(* Logix 5000 project; controller reports 1756-L63 rev 20.15; software revision 20.04; part 14 of 52 *)

        [571].time.Day := 11, [571].time.Hour := 15, [571].time.Minute := 59, [571].time.Second := 59, [572].log_data[0].min := 1.0, [572].log_data[0].max := 1.0, [572].log_data[0].total := 300.0, [572].log_data[0].time := 300.0, [572].log_data[0].valid := 1, [572].log_data[1].valid := 1, [572].log_data[2].valid := 1, [572].log_data[3].valid := 1, [572].log_data[4].valid := 1, [572].log_data[5].valid := 1, [572].log_data[6].valid := 1, [572].log_data[7].valid := 1, [572].log_data[8].valid := 1, [572].log_data[9].valid := 1, [572].log_data[10].valid := 1, [572].log_data[11].valid := 1, [572].log_data[12].valid := 1, [572].log_data[13].valid := 1, [572].log_data[14].valid := 1, [572].log_data[15].valid := 1, [572].log_data[16].valid := 1, [572].log_data[17].valid := 1, [572].log_data[18].valid := 1, [572].log_data[19].valid := 1, [572].time.Year := 2023, [572].time.Month := 1, [572].time.Day := 11, [572].time.Hour := 16, [572].time.Minute := 4, [572].time.Second := 59, [573].log_data[0].min := 1.0, [573].log_data[0].max := 1.0, [573].log_data[0].total := 300.0, [573].log_data[0].time := 300.0, [573].log_data[0].minminute := 5, [573].log_data[0].maxminute := 5, [573].log_data[0].valid := 1, [573].log_data[1].valid := 1, [573].log_data[2].valid := 1, [573].log_data[3].valid := 1, [573].log_data[4].valid := 1, [573].log_data[5].valid := 1, [573].log_data[6].valid := 1, [573].log_data[7].valid := 1, [573].log_data[8].valid := 1, [573].log_data[9].valid := 1, [573].log_data[10].valid := 1, [573].log_data[11].valid := 1, [573].log_data[12].valid := 1, [573].log_data[13].valid := 1, [573].log_data[14].valid := 1, [573].log_data[15].valid := 1, [573].log_data[16].valid := 1, [573].log_data[17].valid := 1, [573].log_data[18].valid := 1, [573].log_data[19].valid := 1,
        [573].time.Year := 2023, [573].time.Month := 1, [573].time.Day := 11, [573].time.Hour := 16, [573].time.Minute := 9, [573].time.Second := 59, [574].log_data[0].min := 1.0, [574].log_data[0].max := 1.0, [574].log_data[0].total := 300.0, [574].log_data[0].time := 300.0, [574].log_data[0].minminute := 10, [574].log_data[0].maxminute := 10, [574].log_data[0].valid := 1, [574].log_data[1].valid := 1, [574].log_data[2].valid := 1, [574].log_data[3].valid := 1, [574].log_data[4].valid := 1, [574].log_data[5].valid := 1, [574].log_data[6].valid := 1, [574].log_data[7].valid := 1, [574].log_data[8].valid := 1, [574].log_data[9].valid := 1, [574].log_data[10].valid := 1, [574].log_data[11].valid := 1, [574].log_data[12].valid := 1, [574].log_data[13].valid := 1, [574].log_data[14].valid := 1, [574].log_data[15].valid := 1, [574].log_data[16].valid := 1, [574].log_data[17].valid := 1, [574].log_data[18].valid := 1, [574].log_data[19].valid := 1, [574].time.Year := 2023, [574].time.Month := 1, [574].time.Day := 11, [574].time.Hour := 16, [574].time.Minute := 14, [574].time.Second := 59, [575].log_data[0].min := 1.0, [575].log_data[0].max := 1.0, [575].log_data[0].total := 300.0, [575].log_data[0].time := 300.0, [575].log_data[0].minminute := 15, [575].log_data[0].maxminute := 15, [575].log_data[0].valid := 1, [575].log_data[1].valid := 1, [575].log_data[2].valid := 1, [575].log_data[3].valid := 1, [575].log_data[4].valid := 1, [575].log_data[5].valid := 1, [575].log_data[6].valid := 1, [575].log_data[7].valid := 1, [575].log_data[8].valid := 1, [575].log_data[9].valid := 1, [575].log_data[10].valid := 1, [575].log_data[11].valid := 1, [575].log_data[12].valid := 1, [575].log_data[13].valid := 1, [575].log_data[14].valid := 1, [575].log_data[15].valid := 1,
        [575].log_data[16].valid := 1, [575].log_data[17].valid := 1, [575].log_data[18].valid := 1, [575].log_data[19].valid := 1, [575].time.Year := 2023, [575].time.Month := 1, [575].time.Day := 11, [575].time.Hour := 16, [575].time.Minute := 19, [575].time.Second := 59, [576].log_data[0].min := 1.0, [576].log_data[0].max := 1.0, [576].log_data[0].total := 300.0, [576].log_data[0].time := 300.0, [576].log_data[0].minminute := 20, [576].log_data[0].maxminute := 20, [576].log_data[0].valid := 1, [576].log_data[1].valid := 1, [576].log_data[2].valid := 1, [576].log_data[3].valid := 1, [576].log_data[4].valid := 1, [576].log_data[5].valid := 1, [576].log_data[6].valid := 1, [576].log_data[7].valid := 1, [576].log_data[8].valid := 1, [576].log_data[9].valid := 1, [576].log_data[10].valid := 1, [576].log_data[11].valid := 1, [576].log_data[12].valid := 1, [576].log_data[13].valid := 1, [576].log_data[14].valid := 1, [576].log_data[15].valid := 1, [576].log_data[16].valid := 1, [576].log_data[17].valid := 1, [576].log_data[18].valid := 1, [576].log_data[19].valid := 1, [576].time.Year := 2023, [576].time.Month := 1, [576].time.Day := 11, [576].time.Hour := 16, [576].time.Minute := 24, [576].time.Second := 59, [577].log_data[0].min := 1.0, [577].log_data[0].max := 1.0, [577].log_data[0].total := 300.0, [577].log_data[0].time := 300.0, [577].log_data[0].minminute := 25, [577].log_data[0].maxminute := 25, [577].log_data[0].valid := 1, [577].log_data[1].valid := 1, [577].log_data[2].valid := 1, [577].log_data[3].valid := 1, [577].log_data[4].valid := 1, [577].log_data[5].valid := 1, [577].log_data[6].valid := 1, [577].log_data[7].valid := 1, [577].log_data[8].valid := 1, [577].log_data[9].valid := 1, [577].log_data[10].valid := 1, [577].log_data[11].valid := 1,
        [577].log_data[12].valid := 1, [577].log_data[13].valid := 1, [577].log_data[14].valid := 1, [577].log_data[15].valid := 1, [577].log_data[16].valid := 1, [577].log_data[17].valid := 1, [577].log_data[18].valid := 1, [577].log_data[19].valid := 1, [577].time.Year := 2023, [577].time.Month := 1, [577].time.Day := 11, [577].time.Hour := 16, [577].time.Minute := 29, [577].time.Second := 59, [578].log_data[0].min := 1.0, [578].log_data[0].max := 1.0, [578].log_data[0].total := 300.0, [578].log_data[0].time := 300.0, [578].log_data[0].minminute := 30, [578].log_data[0].maxminute := 30, [578].log_data[0].valid := 1, [578].log_data[1].valid := 1, [578].log_data[2].valid := 1, [578].log_data[3].valid := 1, [578].log_data[4].valid := 1, [578].log_data[5].valid := 1, [578].log_data[6].valid := 1, [578].log_data[7].valid := 1, [578].log_data[8].valid := 1, [578].log_data[9].valid := 1, [578].log_data[10].valid := 1, [578].log_data[11].valid := 1, [578].log_data[12].valid := 1, [578].log_data[13].valid := 1, [578].log_data[14].valid := 1, [578].log_data[15].valid := 1, [578].log_data[16].valid := 1, [578].log_data[17].valid := 1, [578].log_data[18].valid := 1, [578].log_data[19].valid := 1, [578].time.Year := 2023, [578].time.Month := 1, [578].time.Day := 11, [578].time.Hour := 16, [578].time.Minute := 34, [578].time.Second := 59, [579].log_data[0].min := 1.0, [579].log_data[0].max := 1.0, [579].log_data[0].total := 300.0, [579].log_data[0].time := 300.0, [579].log_data[0].minminute := 35, [579].log_data[0].maxminute := 35, [579].log_data[0].valid := 1, [579].log_data[1].valid := 1, [579].log_data[2].valid := 1, [579].log_data[3].valid := 1, [579].log_data[4].valid := 1, [579].log_data[5].valid := 1, [579].log_data[6].valid := 1, [579].log_data[7].valid := 1,
        [579].log_data[8].valid := 1, [579].log_data[9].valid := 1, [579].log_data[10].valid := 1, [579].log_data[11].valid := 1, [579].log_data[12].valid := 1, [579].log_data[13].valid := 1, [579].log_data[14].valid := 1, [579].log_data[15].valid := 1, [579].log_data[16].valid := 1, [579].log_data[17].valid := 1, [579].log_data[18].valid := 1, [579].log_data[19].valid := 1, [579].time.Year := 2023, [579].time.Month := 1, [579].time.Day := 11, [579].time.Hour := 16, [579].time.Minute := 39, [579].time.Second := 59, [580].log_data[0].min := 1.0, [580].log_data[0].max := 1.0, [580].log_data[0].total := 300.0, [580].log_data[0].time := 300.0, [580].log_data[0].minminute := 40, [580].log_data[0].maxminute := 40, [580].log_data[0].valid := 1, [580].log_data[1].valid := 1, [580].log_data[2].valid := 1, [580].log_data[3].valid := 1, [580].log_data[4].valid := 1, [580].log_data[5].valid := 1, [580].log_data[6].valid := 1, [580].log_data[7].valid := 1, [580].log_data[8].valid := 1, [580].log_data[9].valid := 1, [580].log_data[10].valid := 1, [580].log_data[11].valid := 1, [580].log_data[12].valid := 1, [580].log_data[13].valid := 1, [580].log_data[14].valid := 1, [580].log_data[15].valid := 1, [580].log_data[16].valid := 1, [580].log_data[17].valid := 1, [580].log_data[18].valid := 1, [580].log_data[19].valid := 1, [580].time.Year := 2023, [580].time.Month := 1, [580].time.Day := 11, [580].time.Hour := 16, [580].time.Minute := 44, [580].time.Second := 59, [581].log_data[0].min := 1.0, [581].log_data[0].max := 1.0, [581].log_data[0].total := 300.0, [581].log_data[0].time := 300.0, [581].log_data[0].minminute := 45, [581].log_data[0].maxminute := 45, [581].log_data[0].valid := 1, [581].log_data[1].valid := 1, [581].log_data[2].valid := 1, [581].log_data[3].valid := 1,
        [581].log_data[4].valid := 1, [581].log_data[5].valid := 1, [581].log_data[6].valid := 1, [581].log_data[7].valid := 1, [581].log_data[8].valid := 1, [581].log_data[9].valid := 1, [581].log_data[10].valid := 1, [581].log_data[11].valid := 1, [581].log_data[12].valid := 1, [581].log_data[13].valid := 1, [581].log_data[14].valid := 1, [581].log_data[15].valid := 1, [581].log_data[16].valid := 1, [581].log_data[17].valid := 1, [581].log_data[18].valid := 1, [581].log_data[19].valid := 1, [581].time.Year := 2023, [581].time.Month := 1, [581].time.Day := 11, [581].time.Hour := 16, [581].time.Minute := 49, [581].time.Second := 59, [582].log_data[0].min := 1.0, [582].log_data[0].max := 1.0, [582].log_data[0].total := 300.0, [582].log_data[0].time := 300.0, [582].log_data[0].minminute := 50, [582].log_data[0].maxminute := 50, [582].log_data[0].valid := 1, [582].log_data[1].valid := 1, [582].log_data[2].valid := 1, [582].log_data[3].valid := 1, [582].log_data[4].valid := 1, [582].log_data[5].valid := 1, [582].log_data[6].valid := 1, [582].log_data[7].valid := 1, [582].log_data[8].valid := 1, [582].log_data[9].valid := 1, [582].log_data[10].valid := 1, [582].log_data[11].valid := 1, [582].log_data[12].valid := 1, [582].log_data[13].valid := 1, [582].log_data[14].valid := 1, [582].log_data[15].valid := 1, [582].log_data[16].valid := 1, [582].log_data[17].valid := 1, [582].log_data[18].valid := 1, [582].log_data[19].valid := 1, [582].time.Year := 2023, [582].time.Month := 1, [582].time.Day := 11, [582].time.Hour := 16, [582].time.Minute := 54, [582].time.Second := 59, [583].log_data[0].min := 1.0, [583].log_data[0].max := 1.0, [583].log_data[0].total := 300.0, [583].log_data[0].time := 300.0, [583].log_data[0].minminute := 55, [583].log_data[0].maxminute := 55,
        [583].log_data[0].valid := 1, [583].log_data[1].valid := 1, [583].log_data[2].valid := 1, [583].log_data[3].valid := 1, [583].log_data[4].valid := 1, [583].log_data[5].valid := 1, [583].log_data[6].valid := 1, [583].log_data[7].valid := 1, [583].log_data[8].valid := 1, [583].log_data[9].valid := 1, [583].log_data[10].valid := 1, [583].log_data[11].valid := 1, [583].log_data[12].valid := 1, [583].log_data[13].valid := 1, [583].log_data[14].valid := 1, [583].log_data[15].valid := 1, [583].log_data[16].valid := 1, [583].log_data[17].valid := 1, [583].log_data[18].valid := 1, [583].log_data[19].valid := 1, [583].time.Year := 2023, [583].time.Month := 1, [583].time.Day := 11, [583].time.Hour := 16, [583].time.Minute := 59, [583].time.Second := 59, [584].log_data[0].min := 1.0, [584].log_data[0].max := 1.0, [584].log_data[0].total := 300.0, [584].log_data[0].time := 300.0, [584].log_data[0].valid := 1, [584].log_data[1].valid := 1, [584].log_data[2].valid := 1, [584].log_data[3].valid := 1, [584].log_data[4].valid := 1, [584].log_data[5].valid := 1, [584].log_data[6].valid := 1, [584].log_data[7].valid := 1, [584].log_data[8].valid := 1, [584].log_data[9].valid := 1, [584].log_data[10].valid := 1, [584].log_data[11].valid := 1, [584].log_data[12].valid := 1, [584].log_data[13].valid := 1, [584].log_data[14].valid := 1, [584].log_data[15].valid := 1, [584].log_data[16].valid := 1, [584].log_data[17].valid := 1, [584].log_data[18].valid := 1, [584].log_data[19].valid := 1, [584].time.Year := 2023, [584].time.Month := 1, [584].time.Day := 11, [584].time.Hour := 17, [584].time.Minute := 4, [584].time.Second := 59, [585].log_data[0].min := 1.0, [585].log_data[0].max := 1.0, [585].log_data[0].total := 300.0, [585].log_data[0].time := 300.0,
        [585].log_data[0].minminute := 5, [585].log_data[0].maxminute := 5, [585].log_data[0].valid := 1, [585].log_data[1].valid := 1, [585].log_data[2].valid := 1, [585].log_data[3].valid := 1, [585].log_data[4].valid := 1, [585].log_data[5].valid := 1, [585].log_data[6].valid := 1, [585].log_data[7].valid := 1, [585].log_data[8].valid := 1, [585].log_data[9].valid := 1, [585].log_data[10].valid := 1, [585].log_data[11].valid := 1, [585].log_data[12].valid := 1, [585].log_data[13].valid := 1, [585].log_data[14].valid := 1, [585].log_data[15].valid := 1, [585].log_data[16].valid := 1, [585].log_data[17].valid := 1, [585].log_data[18].valid := 1, [585].log_data[19].valid := 1, [585].time.Year := 2023, [585].time.Month := 1, [585].time.Day := 11, [585].time.Hour := 17, [585].time.Minute := 9, [585].time.Second := 59, [586].log_data[0].min := 1.0, [586].log_data[0].max := 1.0, [586].log_data[0].total := 300.0, [586].log_data[0].time := 300.0, [586].log_data[0].minminute := 10, [586].log_data[0].maxminute := 10, [586].log_data[0].valid := 1, [586].log_data[1].valid := 1, [586].log_data[2].valid := 1, [586].log_data[3].valid := 1, [586].log_data[4].valid := 1, [586].log_data[5].valid := 1, [586].log_data[6].valid := 1, [586].log_data[7].valid := 1, [586].log_data[8].valid := 1, [586].log_data[9].valid := 1, [586].log_data[10].valid := 1, [586].log_data[11].valid := 1, [586].log_data[12].valid := 1, [586].log_data[13].valid := 1, [586].log_data[14].valid := 1, [586].log_data[15].valid := 1, [586].log_data[16].valid := 1, [586].log_data[17].valid := 1, [586].log_data[18].valid := 1, [586].log_data[19].valid := 1, [586].time.Year := 2023, [586].time.Month := 1, [586].time.Day := 11, [586].time.Hour := 17, [586].time.Minute := 14, [586].time.Second := 59,
        [587].log_data[0].min := 1.0, [587].log_data[0].max := 1.0, [587].log_data[0].total := 300.0, [587].log_data[0].time := 300.0, [587].log_data[0].minminute := 15, [587].log_data[0].maxminute := 15, [587].log_data[0].valid := 1, [587].log_data[1].valid := 1, [587].log_data[2].valid := 1, [587].log_data[3].valid := 1, [587].log_data[4].valid := 1, [587].log_data[5].valid := 1, [587].log_data[6].valid := 1, [587].log_data[7].valid := 1, [587].log_data[8].valid := 1, [587].log_data[9].valid := 1, [587].log_data[10].valid := 1, [587].log_data[11].valid := 1, [587].log_data[12].valid := 1, [587].log_data[13].valid := 1, [587].log_data[14].valid := 1, [587].log_data[15].valid := 1, [587].log_data[16].valid := 1, [587].log_data[17].valid := 1, [587].log_data[18].valid := 1, [587].log_data[19].valid := 1, [587].time.Year := 2023, [587].time.Month := 1, [587].time.Day := 11, [587].time.Hour := 17, [587].time.Minute := 19, [587].time.Second := 59, [588].log_data[0].min := 1.0, [588].log_data[0].max := 1.0, [588].log_data[0].total := 300.0, [588].log_data[0].time := 300.0, [588].log_data[0].minminute := 20, [588].log_data[0].maxminute := 20, [588].log_data[0].valid := 1, [588].log_data[1].valid := 1, [588].log_data[2].valid := 1, [588].log_data[3].valid := 1, [588].log_data[4].valid := 1, [588].log_data[5].valid := 1, [588].log_data[6].valid := 1, [588].log_data[7].valid := 1, [588].log_data[8].valid := 1, [588].log_data[9].valid := 1, [588].log_data[10].valid := 1, [588].log_data[11].valid := 1, [588].log_data[12].valid := 1, [588].log_data[13].valid := 1, [588].log_data[14].valid := 1, [588].log_data[15].valid := 1, [588].log_data[16].valid := 1, [588].log_data[17].valid := 1, [588].log_data[18].valid := 1, [588].log_data[19].valid := 1, [588].time.Year := 2023, [588].time.Month := 1,
        [588].time.Day := 11, [588].time.Hour := 17, [588].time.Minute := 24, [588].time.Second := 59, [589].log_data[0].min := 1.0, [589].log_data[0].max := 1.0, [589].log_data[0].total := 300.0, [589].log_data[0].time := 300.0, [589].log_data[0].minminute := 25, [589].log_data[0].maxminute := 25, [589].log_data[0].valid := 1, [589].log_data[1].valid := 1, [589].log_data[2].valid := 1, [589].log_data[3].valid := 1, [589].log_data[4].valid := 1, [589].log_data[5].valid := 1, [589].log_data[6].valid := 1, [589].log_data[7].valid := 1, [589].log_data[8].valid := 1, [589].log_data[9].valid := 1, [589].log_data[10].valid := 1, [589].log_data[11].valid := 1, [589].log_data[12].valid := 1, [589].log_data[13].valid := 1, [589].log_data[14].valid := 1, [589].log_data[15].valid := 1, [589].log_data[16].valid := 1, [589].log_data[17].valid := 1, [589].log_data[18].valid := 1, [589].log_data[19].valid := 1, [589].time.Year := 2023, [589].time.Month := 1, [589].time.Day := 11, [589].time.Hour := 17, [589].time.Minute := 29, [589].time.Second := 59, [590].log_data[0].min := 1.0, [590].log_data[0].max := 1.0, [590].log_data[0].total := 300.0, [590].log_data[0].time := 300.0, [590].log_data[0].minminute := 30, [590].log_data[0].maxminute := 30, [590].log_data[0].valid := 1, [590].log_data[1].valid := 1, [590].log_data[2].valid := 1, [590].log_data[3].valid := 1, [590].log_data[4].valid := 1, [590].log_data[5].valid := 1, [590].log_data[6].valid := 1, [590].log_data[7].valid := 1, [590].log_data[8].valid := 1, [590].log_data[9].valid := 1, [590].log_data[10].valid := 1, [590].log_data[11].valid := 1, [590].log_data[12].valid := 1, [590].log_data[13].valid := 1, [590].log_data[14].valid := 1, [590].log_data[15].valid := 1, [590].log_data[16].valid := 1, [590].log_data[17].valid := 1,
        [590].log_data[18].valid := 1, [590].log_data[19].valid := 1, [590].time.Year := 2023, [590].time.Month := 1, [590].time.Day := 11, [590].time.Hour := 17, [590].time.Minute := 34, [590].time.Second := 59, [591].log_data[0].min := 1.0, [591].log_data[0].max := 1.0, [591].log_data[0].total := 300.0, [591].log_data[0].time := 300.0, [591].log_data[0].minminute := 35, [591].log_data[0].maxminute := 35, [591].log_data[0].valid := 1, [591].log_data[1].valid := 1, [591].log_data[2].valid := 1, [591].log_data[3].valid := 1, [591].log_data[4].valid := 1, [591].log_data[5].valid := 1, [591].log_data[6].valid := 1, [591].log_data[7].valid := 1, [591].log_data[8].valid := 1, [591].log_data[9].valid := 1, [591].log_data[10].valid := 1, [591].log_data[11].valid := 1, [591].log_data[12].valid := 1, [591].log_data[13].valid := 1, [591].log_data[14].valid := 1, [591].log_data[15].valid := 1, [591].log_data[16].valid := 1, [591].log_data[17].valid := 1, [591].log_data[18].valid := 1, [591].log_data[19].valid := 1, [591].time.Year := 2023, [591].time.Month := 1, [591].time.Day := 11, [591].time.Hour := 17, [591].time.Minute := 39, [591].time.Second := 59, [592].log_data[0].min := 1.0, [592].log_data[0].max := 1.0, [592].log_data[0].total := 300.0, [592].log_data[0].time := 300.0, [592].log_data[0].minminute := 40, [592].log_data[0].maxminute := 40, [592].log_data[0].valid := 1, [592].log_data[1].valid := 1, [592].log_data[2].valid := 1, [592].log_data[3].valid := 1, [592].log_data[4].valid := 1, [592].log_data[5].valid := 1, [592].log_data[6].valid := 1, [592].log_data[7].valid := 1, [592].log_data[8].valid := 1, [592].log_data[9].valid := 1, [592].log_data[10].valid := 1, [592].log_data[11].valid := 1, [592].log_data[12].valid := 1, [592].log_data[13].valid := 1,
        [592].log_data[14].valid := 1, [592].log_data[15].valid := 1, [592].log_data[16].valid := 1, [592].log_data[17].valid := 1, [592].log_data[18].valid := 1, [592].log_data[19].valid := 1, [592].time.Year := 2023, [592].time.Month := 1, [592].time.Day := 11, [592].time.Hour := 17, [592].time.Minute := 44, [592].time.Second := 59, [593].log_data[0].min := 1.0, [593].log_data[0].max := 1.0, [593].log_data[0].total := 300.0, [593].log_data[0].time := 300.0, [593].log_data[0].minminute := 45, [593].log_data[0].maxminute := 45, [593].log_data[0].valid := 1, [593].log_data[1].valid := 1, [593].log_data[2].valid := 1, [593].log_data[3].valid := 1, [593].log_data[4].valid := 1, [593].log_data[5].valid := 1, [593].log_data[6].valid := 1, [593].log_data[7].valid := 1, [593].log_data[8].valid := 1, [593].log_data[9].valid := 1, [593].log_data[10].valid := 1, [593].log_data[11].valid := 1, [593].log_data[12].valid := 1, [593].log_data[13].valid := 1, [593].log_data[14].valid := 1, [593].log_data[15].valid := 1, [593].log_data[16].valid := 1, [593].log_data[17].valid := 1, [593].log_data[18].valid := 1, [593].log_data[19].valid := 1, [593].time.Year := 2023, [593].time.Month := 1, [593].time.Day := 11, [593].time.Hour := 17, [593].time.Minute := 49, [593].time.Second := 59, [594].log_data[0].min := 1.0, [594].log_data[0].max := 1.0, [594].log_data[0].total := 300.0, [594].log_data[0].time := 300.0, [594].log_data[0].minminute := 50, [594].log_data[0].maxminute := 50, [594].log_data[0].valid := 1, [594].log_data[1].valid := 1, [594].log_data[2].valid := 1, [594].log_data[3].valid := 1, [594].log_data[4].valid := 1, [594].log_data[5].valid := 1, [594].log_data[6].valid := 1, [594].log_data[7].valid := 1, [594].log_data[8].valid := 1, [594].log_data[9].valid := 1,
        [594].log_data[10].valid := 1, [594].log_data[11].valid := 1, [594].log_data[12].valid := 1, [594].log_data[13].valid := 1, [594].log_data[14].valid := 1, [594].log_data[15].valid := 1, [594].log_data[16].valid := 1, [594].log_data[17].valid := 1, [594].log_data[18].valid := 1, [594].log_data[19].valid := 1, [594].time.Year := 2023, [594].time.Month := 1, [594].time.Day := 11, [594].time.Hour := 17, [594].time.Minute := 54, [594].time.Second := 59, [595].log_data[0].min := 1.0, [595].log_data[0].max := 1.0, [595].log_data[0].total := 300.0, [595].log_data[0].time := 300.0, [595].log_data[0].minminute := 55, [595].log_data[0].maxminute := 55, [595].log_data[0].valid := 1, [595].log_data[1].valid := 1, [595].log_data[2].valid := 1, [595].log_data[3].valid := 1, [595].log_data[4].valid := 1, [595].log_data[5].valid := 1, [595].log_data[6].valid := 1, [595].log_data[7].valid := 1, [595].log_data[8].valid := 1, [595].log_data[9].valid := 1, [595].log_data[10].valid := 1, [595].log_data[11].valid := 1, [595].log_data[12].valid := 1, [595].log_data[13].valid := 1, [595].log_data[14].valid := 1, [595].log_data[15].valid := 1, [595].log_data[16].valid := 1, [595].log_data[17].valid := 1, [595].log_data[18].valid := 1, [595].log_data[19].valid := 1, [595].time.Year := 2023, [595].time.Month := 1, [595].time.Day := 11, [595].time.Hour := 17, [595].time.Minute := 59, [595].time.Second := 59, [596].log_data[0].min := 1.0, [596].log_data[0].max := 1.0, [596].log_data[0].total := 300.0, [596].log_data[0].time := 300.0, [596].log_data[0].valid := 1, [596].log_data[1].valid := 1, [596].log_data[2].valid := 1, [596].log_data[3].valid := 1, [596].log_data[4].valid := 1, [596].log_data[5].valid := 1, [596].log_data[6].valid := 1, [596].log_data[7].valid := 1,
        [596].log_data[8].valid := 1, [596].log_data[9].valid := 1, [596].log_data[10].valid := 1, [596].log_data[11].valid := 1, [596].log_data[12].valid := 1, [596].log_data[13].valid := 1, [596].log_data[14].valid := 1, [596].log_data[15].valid := 1, [596].log_data[16].valid := 1, [596].log_data[17].valid := 1, [596].log_data[18].valid := 1, [596].log_data[19].valid := 1, [596].time.Year := 2023, [596].time.Month := 1, [596].time.Day := 11, [596].time.Hour := 18, [596].time.Minute := 4, [596].time.Second := 59, [597].log_data[0].min := 1.0, [597].log_data[0].max := 1.0, [597].log_data[0].total := 300.0, [597].log_data[0].time := 300.0, [597].log_data[0].minminute := 5, [597].log_data[0].maxminute := 5, [597].log_data[0].valid := 1, [597].log_data[1].valid := 1, [597].log_data[2].valid := 1, [597].log_data[3].valid := 1, [597].log_data[4].valid := 1, [597].log_data[5].valid := 1, [597].log_data[6].valid := 1, [597].log_data[7].valid := 1, [597].log_data[8].valid := 1, [597].log_data[9].valid := 1, [597].log_data[10].valid := 1, [597].log_data[11].valid := 1, [597].log_data[12].valid := 1, [597].log_data[13].valid := 1, [597].log_data[14].valid := 1, [597].log_data[15].valid := 1, [597].log_data[16].valid := 1, [597].log_data[17].valid := 1, [597].log_data[18].valid := 1, [597].log_data[19].valid := 1, [597].time.Year := 2023, [597].time.Month := 1, [597].time.Day := 11, [597].time.Hour := 18, [597].time.Minute := 9, [597].time.Second := 59, [598].log_data[0].min := 1.0, [598].log_data[0].max := 1.0, [598].log_data[0].total := 300.0, [598].log_data[0].time := 300.0, [598].log_data[0].minminute := 10, [598].log_data[0].maxminute := 10, [598].log_data[0].valid := 1, [598].log_data[1].valid := 1, [598].log_data[2].valid := 1, [598].log_data[3].valid := 1,
        [598].log_data[4].valid := 1, [598].log_data[5].valid := 1, [598].log_data[6].valid := 1, [598].log_data[7].valid := 1, [598].log_data[8].valid := 1, [598].log_data[9].valid := 1, [598].log_data[10].valid := 1, [598].log_data[11].valid := 1, [598].log_data[12].valid := 1, [598].log_data[13].valid := 1, [598].log_data[14].valid := 1, [598].log_data[15].valid := 1, [598].log_data[16].valid := 1, [598].log_data[17].valid := 1, [598].log_data[18].valid := 1, [598].log_data[19].valid := 1, [598].time.Year := 2023, [598].time.Month := 1, [598].time.Day := 11, [598].time.Hour := 18, [598].time.Minute := 14, [598].time.Second := 59, [599].log_data[0].min := 1.0, [599].log_data[0].max := 1.0, [599].log_data[0].total := 300.0, [599].log_data[0].time := 300.0, [599].log_data[0].minminute := 15, [599].log_data[0].maxminute := 15, [599].log_data[0].valid := 1, [599].log_data[1].valid := 1, [599].log_data[2].valid := 1, [599].log_data[3].valid := 1, [599].log_data[4].valid := 1, [599].log_data[5].valid := 1, [599].log_data[6].valid := 1, [599].log_data[7].valid := 1, [599].log_data[8].valid := 1, [599].log_data[9].valid := 1, [599].log_data[10].valid := 1, [599].log_data[11].valid := 1, [599].log_data[12].valid := 1, [599].log_data[13].valid := 1, [599].log_data[14].valid := 1, [599].log_data[15].valid := 1, [599].log_data[16].valid := 1, [599].log_data[17].valid := 1, [599].log_data[18].valid := 1, [599].log_data[19].valid := 1, [599].time.Year := 2023, [599].time.Month := 1, [599].time.Day := 11, [599].time.Hour := 18, [599].time.Minute := 19, [599].time.Second := 59, [600].log_data[0].min := 1.0, [600].log_data[0].max := 1.0, [600].log_data[0].total := 300.0, [600].log_data[0].time := 300.0, [600].log_data[0].minminute := 20, [600].log_data[0].maxminute := 20,
        [600].log_data[0].valid := 1, [600].log_data[1].valid := 1, [600].log_data[2].valid := 1, [600].log_data[3].valid := 1, [600].log_data[4].valid := 1, [600].log_data[5].valid := 1, [600].log_data[6].valid := 1, [600].log_data[7].valid := 1, [600].log_data[8].valid := 1, [600].log_data[9].valid := 1, [600].log_data[10].valid := 1, [600].log_data[11].valid := 1, [600].log_data[12].valid := 1, [600].log_data[13].valid := 1, [600].log_data[14].valid := 1, [600].log_data[15].valid := 1, [600].log_data[16].valid := 1, [600].log_data[17].valid := 1, [600].log_data[18].valid := 1, [600].log_data[19].valid := 1, [600].time.Year := 2023, [600].time.Month := 1, [600].time.Day := 11, [600].time.Hour := 18, [600].time.Minute := 24, [600].time.Second := 59, [601].log_data[0].min := 1.0, [601].log_data[0].max := 1.0, [601].log_data[0].total := 300.0, [601].log_data[0].time := 300.0, [601].log_data[0].minminute := 25, [601].log_data[0].maxminute := 25, [601].log_data[0].valid := 1, [601].log_data[1].valid := 1, [601].log_data[2].valid := 1, [601].log_data[3].valid := 1, [601].log_data[4].valid := 1, [601].log_data[5].valid := 1, [601].log_data[6].valid := 1, [601].log_data[7].valid := 1, [601].log_data[8].valid := 1, [601].log_data[9].valid := 1, [601].log_data[10].valid := 1, [601].log_data[11].valid := 1, [601].log_data[12].valid := 1, [601].log_data[13].valid := 1, [601].log_data[14].valid := 1, [601].log_data[15].valid := 1, [601].log_data[16].valid := 1, [601].log_data[17].valid := 1, [601].log_data[18].valid := 1, [601].log_data[19].valid := 1, [601].time.Year := 2023, [601].time.Month := 1, [601].time.Day := 11, [601].time.Hour := 18, [601].time.Minute := 29, [601].time.Second := 59, [602].log_data[0].min := 1.0, [602].log_data[0].max := 1.0,
        [602].log_data[0].total := 300.0, [602].log_data[0].time := 300.0, [602].log_data[0].minminute := 30, [602].log_data[0].maxminute := 30, [602].log_data[0].valid := 1, [602].log_data[1].valid := 1, [602].log_data[2].valid := 1, [602].log_data[3].valid := 1, [602].log_data[4].valid := 1, [602].log_data[5].valid := 1, [602].log_data[6].valid := 1, [602].log_data[7].valid := 1, [602].log_data[8].valid := 1, [602].log_data[9].valid := 1, [602].log_data[10].valid := 1, [602].log_data[11].valid := 1, [602].log_data[12].valid := 1, [602].log_data[13].valid := 1, [602].log_data[14].valid := 1, [602].log_data[15].valid := 1, [602].log_data[16].valid := 1, [602].log_data[17].valid := 1, [602].log_data[18].valid := 1, [602].log_data[19].valid := 1, [602].time.Year := 2023, [602].time.Month := 1, [602].time.Day := 11, [602].time.Hour := 18, [602].time.Minute := 34, [602].time.Second := 59, [603].log_data[0].min := 1.0, [603].log_data[0].max := 1.0, [603].log_data[0].total := 300.0, [603].log_data[0].time := 300.0, [603].log_data[0].minminute := 35, [603].log_data[0].maxminute := 35, [603].log_data[0].valid := 1, [603].log_data[1].valid := 1, [603].log_data[2].valid := 1, [603].log_data[3].valid := 1, [603].log_data[4].valid := 1, [603].log_data[5].valid := 1, [603].log_data[6].valid := 1, [603].log_data[7].valid := 1, [603].log_data[8].valid := 1, [603].log_data[9].valid := 1, [603].log_data[10].valid := 1, [603].log_data[11].valid := 1, [603].log_data[12].valid := 1, [603].log_data[13].valid := 1, [603].log_data[14].valid := 1, [603].log_data[15].valid := 1, [603].log_data[16].valid := 1, [603].log_data[17].valid := 1, [603].log_data[18].valid := 1, [603].log_data[19].valid := 1, [603].time.Year := 2023, [603].time.Month := 1, [603].time.Day := 11, [603].time.Hour := 18,
        [603].time.Minute := 39, [603].time.Second := 59, [604].log_data[0].min := 1.0, [604].log_data[0].max := 1.0, [604].log_data[0].total := 300.0, [604].log_data[0].time := 300.0, [604].log_data[0].minminute := 40, [604].log_data[0].maxminute := 40, [604].log_data[0].valid := 1, [604].log_data[1].valid := 1, [604].log_data[2].valid := 1, [604].log_data[3].valid := 1, [604].log_data[4].valid := 1, [604].log_data[5].valid := 1, [604].log_data[6].valid := 1, [604].log_data[7].valid := 1, [604].log_data[8].valid := 1, [604].log_data[9].valid := 1, [604].log_data[10].valid := 1, [604].log_data[11].valid := 1, [604].log_data[12].valid := 1, [604].log_data[13].valid := 1, [604].log_data[14].valid := 1, [604].log_data[15].valid := 1, [604].log_data[16].valid := 1, [604].log_data[17].valid := 1, [604].log_data[18].valid := 1, [604].log_data[19].valid := 1, [604].time.Year := 2023, [604].time.Month := 1, [604].time.Day := 11, [604].time.Hour := 18, [604].time.Minute := 44, [604].time.Second := 59, [605].log_data[0].min := 1.0, [605].log_data[0].max := 1.0, [605].log_data[0].total := 300.0, [605].log_data[0].time := 300.0, [605].log_data[0].minminute := 45, [605].log_data[0].maxminute := 45, [605].log_data[0].valid := 1, [605].log_data[1].valid := 1, [605].log_data[2].valid := 1, [605].log_data[3].valid := 1, [605].log_data[4].valid := 1, [605].log_data[5].valid := 1, [605].log_data[6].valid := 1, [605].log_data[7].valid := 1, [605].log_data[8].valid := 1, [605].log_data[9].valid := 1, [605].log_data[10].valid := 1, [605].log_data[11].valid := 1, [605].log_data[12].valid := 1, [605].log_data[13].valid := 1, [605].log_data[14].valid := 1, [605].log_data[15].valid := 1, [605].log_data[16].valid := 1, [605].log_data[17].valid := 1, [605].log_data[18].valid := 1, [605].log_data[19].valid := 1,
        [605].time.Year := 2023, [605].time.Month := 1, [605].time.Day := 11, [605].time.Hour := 18, [605].time.Minute := 49, [605].time.Second := 59, [606].log_data[0].min := 1.0, [606].log_data[0].max := 1.0, [606].log_data[0].total := 300.0, [606].log_data[0].time := 300.0, [606].log_data[0].minminute := 50, [606].log_data[0].maxminute := 50, [606].log_data[0].valid := 1, [606].log_data[1].valid := 1, [606].log_data[2].valid := 1, [606].log_data[3].valid := 1, [606].log_data[4].valid := 1, [606].log_data[5].valid := 1, [606].log_data[6].valid := 1, [606].log_data[7].valid := 1, [606].log_data[8].valid := 1, [606].log_data[9].valid := 1, [606].log_data[10].valid := 1, [606].log_data[11].valid := 1, [606].log_data[12].valid := 1, [606].log_data[13].valid := 1, [606].log_data[14].valid := 1, [606].log_data[15].valid := 1, [606].log_data[16].valid := 1, [606].log_data[17].valid := 1, [606].log_data[18].valid := 1, [606].log_data[19].valid := 1, [606].time.Year := 2023, [606].time.Month := 1, [606].time.Day := 11, [606].time.Hour := 18, [606].time.Minute := 54, [606].time.Second := 59, [607].log_data[0].min := 1.0, [607].log_data[0].max := 1.0, [607].log_data[0].total := 300.0, [607].log_data[0].time := 300.0, [607].log_data[0].minminute := 55, [607].log_data[0].maxminute := 55, [607].log_data[0].valid := 1, [607].log_data[1].valid := 1, [607].log_data[2].valid := 1, [607].log_data[3].valid := 1, [607].log_data[4].valid := 1, [607].log_data[5].valid := 1, [607].log_data[6].valid := 1, [607].log_data[7].valid := 1, [607].log_data[8].valid := 1, [607].log_data[9].valid := 1, [607].log_data[10].valid := 1, [607].log_data[11].valid := 1, [607].log_data[12].valid := 1, [607].log_data[13].valid := 1, [607].log_data[14].valid := 1, [607].log_data[15].valid := 1,
        [607].log_data[16].valid := 1, [607].log_data[17].valid := 1, [607].log_data[18].valid := 1, [607].log_data[19].valid := 1, [607].time.Year := 2023, [607].time.Month := 1, [607].time.Day := 11, [607].time.Hour := 18, [607].time.Minute := 59, [607].time.Second := 59, [608].log_data[0].min := 1.0, [608].log_data[0].max := 1.0, [608].log_data[0].total := 300.0, [608].log_data[0].time := 300.0, [608].log_data[0].valid := 1, [608].log_data[1].valid := 1, [608].log_data[2].valid := 1, [608].log_data[3].valid := 1, [608].log_data[4].valid := 1, [608].log_data[5].valid := 1, [608].log_data[6].valid := 1, [608].log_data[7].valid := 1, [608].log_data[8].valid := 1, [608].log_data[9].valid := 1, [608].log_data[10].valid := 1, [608].log_data[11].valid := 1, [608].log_data[12].valid := 1, [608].log_data[13].valid := 1, [608].log_data[14].valid := 1, [608].log_data[15].valid := 1, [608].log_data[16].valid := 1, [608].log_data[17].valid := 1, [608].log_data[18].valid := 1, [608].log_data[19].valid := 1, [608].time.Year := 2023, [608].time.Month := 1, [608].time.Day := 11, [608].time.Hour := 19, [608].time.Minute := 4, [608].time.Second := 59, [609].log_data[0].min := 1.0, [609].log_data[0].max := 1.0, [609].log_data[0].total := 300.0, [609].log_data[0].time := 300.0, [609].log_data[0].minminute := 5, [609].log_data[0].maxminute := 5, [609].log_data[0].valid := 1, [609].log_data[1].valid := 1, [609].log_data[2].valid := 1, [609].log_data[3].valid := 1, [609].log_data[4].valid := 1, [609].log_data[5].valid := 1, [609].log_data[6].valid := 1, [609].log_data[7].valid := 1, [609].log_data[8].valid := 1, [609].log_data[9].valid := 1, [609].log_data[10].valid := 1, [609].log_data[11].valid := 1, [609].log_data[12].valid := 1, [609].log_data[13].valid := 1,
        [609].log_data[14].valid := 1, [609].log_data[15].valid := 1, [609].log_data[16].valid := 1, [609].log_data[17].valid := 1, [609].log_data[18].valid := 1, [609].log_data[19].valid := 1, [609].time.Year := 2023, [609].time.Month := 1, [609].time.Day := 11, [609].time.Hour := 19, [609].time.Minute := 9, [609].time.Second := 59, [610].log_data[0].min := 1.0, [610].log_data[0].max := 1.0, [610].log_data[0].total := 300.0, [610].log_data[0].time := 300.0, [610].log_data[0].minminute := 10, [610].log_data[0].maxminute := 10, [610].log_data[0].valid := 1, [610].log_data[1].valid := 1, [610].log_data[2].valid := 1, [610].log_data[3].valid := 1, [610].log_data[4].valid := 1, [610].log_data[5].valid := 1, [610].log_data[6].valid := 1, [610].log_data[7].valid := 1, [610].log_data[8].valid := 1, [610].log_data[9].valid := 1, [610].log_data[10].valid := 1, [610].log_data[11].valid := 1, [610].log_data[12].valid := 1, [610].log_data[13].valid := 1, [610].log_data[14].valid := 1, [610].log_data[15].valid := 1, [610].log_data[16].valid := 1, [610].log_data[17].valid := 1, [610].log_data[18].valid := 1, [610].log_data[19].valid := 1, [610].time.Year := 2023, [610].time.Month := 1, [610].time.Day := 11, [610].time.Hour := 19, [610].time.Minute := 14, [610].time.Second := 59, [611].log_data[0].min := 1.0, [611].log_data[0].max := 1.0, [611].log_data[0].total := 300.0, [611].log_data[0].time := 300.0, [611].log_data[0].minminute := 15, [611].log_data[0].maxminute := 15, [611].log_data[0].valid := 1, [611].log_data[1].valid := 1, [611].log_data[2].valid := 1, [611].log_data[3].valid := 1, [611].log_data[4].valid := 1, [611].log_data[5].valid := 1, [611].log_data[6].valid := 1, [611].log_data[7].valid := 1, [611].log_data[8].valid := 1, [611].log_data[9].valid := 1,
        [611].log_data[10].valid := 1, [611].log_data[11].valid := 1, [611].log_data[12].valid := 1, [611].log_data[13].valid := 1, [611].log_data[14].valid := 1, [611].log_data[15].valid := 1, [611].log_data[16].valid := 1, [611].log_data[17].valid := 1, [611].log_data[18].valid := 1, [611].log_data[19].valid := 1, [611].time.Year := 2023, [611].time.Month := 1, [611].time.Day := 11, [611].time.Hour := 19, [611].time.Minute := 19, [611].time.Second := 59, [612].log_data[0].min := 1.0, [612].log_data[0].max := 1.0, [612].log_data[0].total := 300.0, [612].log_data[0].time := 300.0, [612].log_data[0].minminute := 20, [612].log_data[0].maxminute := 20, [612].log_data[0].valid := 1, [612].log_data[1].valid := 1, [612].log_data[2].valid := 1, [612].log_data[3].valid := 1, [612].log_data[4].valid := 1, [612].log_data[5].valid := 1, [612].log_data[6].valid := 1, [612].log_data[7].valid := 1, [612].log_data[8].valid := 1, [612].log_data[9].valid := 1, [612].log_data[10].valid := 1, [612].log_data[11].valid := 1, [612].log_data[12].valid := 1, [612].log_data[13].valid := 1, [612].log_data[14].valid := 1, [612].log_data[15].valid := 1, [612].log_data[16].valid := 1, [612].log_data[17].valid := 1, [612].log_data[18].valid := 1, [612].log_data[19].valid := 1, [612].time.Year := 2023, [612].time.Month := 1, [612].time.Day := 11, [612].time.Hour := 19, [612].time.Minute := 24, [612].time.Second := 59, [613].log_data[0].min := 1.0, [613].log_data[0].max := 1.0, [613].log_data[0].total := 300.0, [613].log_data[0].time := 300.0, [613].log_data[0].minminute := 25, [613].log_data[0].maxminute := 25, [613].log_data[0].valid := 1, [613].log_data[1].valid := 1, [613].log_data[2].valid := 1, [613].log_data[3].valid := 1, [613].log_data[4].valid := 1, [613].log_data[5].valid := 1,
        [613].log_data[6].valid := 1, [613].log_data[7].valid := 1, [613].log_data[8].valid := 1, [613].log_data[9].valid := 1, [613].log_data[10].valid := 1, [613].log_data[11].valid := 1, [613].log_data[12].valid := 1, [613].log_data[13].valid := 1, [613].log_data[14].valid := 1, [613].log_data[15].valid := 1, [613].log_data[16].valid := 1, [613].log_data[17].valid := 1, [613].log_data[18].valid := 1, [613].log_data[19].valid := 1, [613].time.Year := 2023, [613].time.Month := 1, [613].time.Day := 11, [613].time.Hour := 19, [613].time.Minute := 29, [613].time.Second := 59, [614].log_data[0].min := 1.0, [614].log_data[0].max := 1.0, [614].log_data[0].total := 300.0, [614].log_data[0].time := 300.0, [614].log_data[0].minminute := 30, [614].log_data[0].maxminute := 30, [614].log_data[0].valid := 1, [614].log_data[1].valid := 1, [614].log_data[2].valid := 1, [614].log_data[3].valid := 1, [614].log_data[4].valid := 1, [614].log_data[5].valid := 1, [614].log_data[6].valid := 1, [614].log_data[7].valid := 1, [614].log_data[8].valid := 1, [614].log_data[9].valid := 1, [614].log_data[10].valid := 1, [614].log_data[11].valid := 1, [614].log_data[12].valid := 1, [614].log_data[13].valid := 1, [614].log_data[14].valid := 1, [614].log_data[15].valid := 1, [614].log_data[16].valid := 1, [614].log_data[17].valid := 1, [614].log_data[18].valid := 1, [614].log_data[19].valid := 1, [614].time.Year := 2023, [614].time.Month := 1, [614].time.Day := 11, [614].time.Hour := 19, [614].time.Minute := 34, [614].time.Second := 59, [615].log_data[0].min := 1.0, [615].log_data[0].max := 1.0, [615].log_data[0].total := 300.0, [615].log_data[0].time := 300.0, [615].log_data[0].minminute := 35, [615].log_data[0].maxminute := 35, [615].log_data[0].valid := 1, [615].log_data[1].valid := 1,
        [615].log_data[2].valid := 1, [615].log_data[3].valid := 1, [615].log_data[4].valid := 1, [615].log_data[5].valid := 1, [615].log_data[6].valid := 1, [615].log_data[7].valid := 1, [615].log_data[8].valid := 1, [615].log_data[9].valid := 1, [615].log_data[10].valid := 1, [615].log_data[11].valid := 1, [615].log_data[12].valid := 1, [615].log_data[13].valid := 1, [615].log_data[14].valid := 1, [615].log_data[15].valid := 1, [615].log_data[16].valid := 1, [615].log_data[17].valid := 1, [615].log_data[18].valid := 1, [615].log_data[19].valid := 1, [615].time.Year := 2023, [615].time.Month := 1, [615].time.Day := 11, [615].time.Hour := 19, [615].time.Minute := 39, [615].time.Second := 59, [616].log_data[0].min := 1.0, [616].log_data[0].max := 1.0, [616].log_data[0].total := 300.0, [616].log_data[0].time := 300.0, [616].log_data[0].minminute := 40, [616].log_data[0].maxminute := 40, [616].log_data[0].valid := 1, [616].log_data[1].valid := 1, [616].log_data[2].valid := 1, [616].log_data[3].valid := 1, [616].log_data[4].valid := 1, [616].log_data[5].valid := 1, [616].log_data[6].valid := 1, [616].log_data[7].valid := 1, [616].log_data[8].valid := 1, [616].log_data[9].valid := 1, [616].log_data[10].valid := 1, [616].log_data[11].valid := 1, [616].log_data[12].valid := 1, [616].log_data[13].valid := 1, [616].log_data[14].valid := 1, [616].log_data[15].valid := 1, [616].log_data[16].valid := 1, [616].log_data[17].valid := 1, [616].log_data[18].valid := 1, [616].log_data[19].valid := 1, [616].time.Year := 2023, [616].time.Month := 1, [616].time.Day := 11, [616].time.Hour := 19, [616].time.Minute := 44, [616].time.Second := 59, [617].log_data[0].min := 1.0, [617].log_data[0].max := 1.0, [617].log_data[0].total := 300.0, [617].log_data[0].time := 300.0,
        [617].log_data[0].minminute := 45, [617].log_data[0].maxminute := 45, [617].log_data[0].valid := 1, [617].log_data[1].valid := 1, [617].log_data[2].valid := 1, [617].log_data[3].valid := 1, [617].log_data[4].valid := 1, [617].log_data[5].valid := 1, [617].log_data[6].valid := 1, [617].log_data[7].valid := 1, [617].log_data[8].valid := 1, [617].log_data[9].valid := 1, [617].log_data[10].valid := 1, [617].log_data[11].valid := 1, [617].log_data[12].valid := 1, [617].log_data[13].valid := 1, [617].log_data[14].valid := 1, [617].log_data[15].valid := 1, [617].log_data[16].valid := 1, [617].log_data[17].valid := 1, [617].log_data[18].valid := 1, [617].log_data[19].valid := 1, [617].time.Year := 2023, [617].time.Month := 1, [617].time.Day := 11, [617].time.Hour := 19, [617].time.Minute := 49, [617].time.Second := 59, [618].log_data[0].min := 1.0, [618].log_data[0].max := 1.0, [618].log_data[0].total := 300.0, [618].log_data[0].time := 300.0, [618].log_data[0].minminute := 50, [618].log_data[0].maxminute := 50, [618].log_data[0].valid := 1, [618].log_data[1].valid := 1, [618].log_data[2].valid := 1, [618].log_data[3].valid := 1, [618].log_data[4].valid := 1, [618].log_data[5].valid := 1, [618].log_data[6].valid := 1, [618].log_data[7].valid := 1, [618].log_data[8].valid := 1, [618].log_data[9].valid := 1, [618].log_data[10].valid := 1, [618].log_data[11].valid := 1, [618].log_data[12].valid := 1, [618].log_data[13].valid := 1, [618].log_data[14].valid := 1, [618].log_data[15].valid := 1, [618].log_data[16].valid := 1, [618].log_data[17].valid := 1, [618].log_data[18].valid := 1, [618].log_data[19].valid := 1, [618].time.Year := 2023, [618].time.Month := 1, [618].time.Day := 11, [618].time.Hour := 19, [618].time.Minute := 54, [618].time.Second := 59,
        [619].log_data[0].min := 1.0, [619].log_data[0].max := 1.0, [619].log_data[0].total := 300.0, [619].log_data[0].time := 300.0, [619].log_data[0].minminute := 55, [619].log_data[0].maxminute := 55, [619].log_data[0].valid := 1, [619].log_data[1].valid := 1, [619].log_data[2].valid := 1, [619].log_data[3].valid := 1, [619].log_data[4].valid := 1, [619].log_data[5].valid := 1, [619].log_data[6].valid := 1, [619].log_data[7].valid := 1, [619].log_data[8].valid := 1, [619].log_data[9].valid := 1, [619].log_data[10].valid := 1, [619].log_data[11].valid := 1, [619].log_data[12].valid := 1, [619].log_data[13].valid := 1, [619].log_data[14].valid := 1, [619].log_data[15].valid := 1, [619].log_data[16].valid := 1, [619].log_data[17].valid := 1, [619].log_data[18].valid := 1, [619].log_data[19].valid := 1, [619].time.Year := 2023, [619].time.Month := 1, [619].time.Day := 11, [619].time.Hour := 19, [619].time.Minute := 59, [619].time.Second := 59, [620].log_data[0].min := 1.0, [620].log_data[0].max := 1.0, [620].log_data[0].total := 300.0, [620].log_data[0].time := 300.0, [620].log_data[0].valid := 1, [620].log_data[1].valid := 1, [620].log_data[2].valid := 1, [620].log_data[3].valid := 1, [620].log_data[4].valid := 1, [620].log_data[5].valid := 1, [620].log_data[6].valid := 1, [620].log_data[7].valid := 1, [620].log_data[8].valid := 1, [620].log_data[9].valid := 1, [620].log_data[10].valid := 1, [620].log_data[11].valid := 1, [620].log_data[12].valid := 1, [620].log_data[13].valid := 1, [620].log_data[14].valid := 1, [620].log_data[15].valid := 1, [620].log_data[16].valid := 1, [620].log_data[17].valid := 1, [620].log_data[18].valid := 1, [620].log_data[19].valid := 1, [620].time.Year := 2023, [620].time.Month := 1, [620].time.Day := 11, [620].time.Hour := 20,
        [620].time.Minute := 4, [620].time.Second := 59, [621].log_data[0].min := 1.0, [621].log_data[0].max := 1.0, [621].log_data[0].total := 300.0, [621].log_data[0].time := 300.0, [621].log_data[0].minminute := 5, [621].log_data[0].maxminute := 5, [621].log_data[0].valid := 1, [621].log_data[1].valid := 1, [621].log_data[2].valid := 1, [621].log_data[3].valid := 1, [621].log_data[4].valid := 1, [621].log_data[5].valid := 1, [621].log_data[6].valid := 1, [621].log_data[7].valid := 1, [621].log_data[8].valid := 1, [621].log_data[9].valid := 1, [621].log_data[10].valid := 1, [621].log_data[11].valid := 1, [621].log_data[12].valid := 1, [621].log_data[13].valid := 1, [621].log_data[14].valid := 1, [621].log_data[15].valid := 1, [621].log_data[16].valid := 1, [621].log_data[17].valid := 1, [621].log_data[18].valid := 1, [621].log_data[19].valid := 1, [621].time.Year := 2023, [621].time.Month := 1, [621].time.Day := 11, [621].time.Hour := 20, [621].time.Minute := 9, [621].time.Second := 59, [622].log_data[0].min := 1.0, [622].log_data[0].max := 1.0, [622].log_data[0].total := 300.0, [622].log_data[0].time := 300.0, [622].log_data[0].minminute := 10, [622].log_data[0].maxminute := 10, [622].log_data[0].valid := 1, [622].log_data[1].valid := 1, [622].log_data[2].valid := 1, [622].log_data[3].valid := 1, [622].log_data[4].valid := 1, [622].log_data[5].valid := 1, [622].log_data[6].valid := 1, [622].log_data[7].valid := 1, [622].log_data[8].valid := 1, [622].log_data[9].valid := 1, [622].log_data[10].valid := 1, [622].log_data[11].valid := 1, [622].log_data[12].valid := 1, [622].log_data[13].valid := 1, [622].log_data[14].valid := 1, [622].log_data[15].valid := 1, [622].log_data[16].valid := 1, [622].log_data[17].valid := 1, [622].log_data[18].valid := 1, [622].log_data[19].valid := 1,
        [622].time.Year := 2023, [622].time.Month := 1, [622].time.Day := 11, [622].time.Hour := 20, [622].time.Minute := 14, [622].time.Second := 59, [623].log_data[0].min := 1.0, [623].log_data[0].max := 1.0, [623].log_data[0].total := 300.0, [623].log_data[0].time := 300.0, [623].log_data[0].minminute := 15, [623].log_data[0].maxminute := 15, [623].log_data[0].valid := 1, [623].log_data[1].valid := 1, [623].log_data[2].valid := 1, [623].log_data[3].valid := 1, [623].log_data[4].valid := 1, [623].log_data[5].valid := 1, [623].log_data[6].valid := 1, [623].log_data[7].valid := 1, [623].log_data[8].valid := 1, [623].log_data[9].valid := 1, [623].log_data[10].valid := 1, [623].log_data[11].valid := 1, [623].log_data[12].valid := 1, [623].log_data[13].valid := 1, [623].log_data[14].valid := 1, [623].log_data[15].valid := 1, [623].log_data[16].valid := 1, [623].log_data[17].valid := 1, [623].log_data[18].valid := 1, [623].log_data[19].valid := 1, [623].time.Year := 2023, [623].time.Month := 1, [623].time.Day := 11, [623].time.Hour := 20, [623].time.Minute := 19, [623].time.Second := 59, [624].log_data[0].min := 1.0, [624].log_data[0].max := 1.0, [624].log_data[0].total := 300.0, [624].log_data[0].time := 300.0, [624].log_data[0].minminute := 20, [624].log_data[0].maxminute := 20, [624].log_data[0].valid := 1, [624].log_data[1].valid := 1, [624].log_data[2].valid := 1, [624].log_data[3].valid := 1, [624].log_data[4].valid := 1, [624].log_data[5].valid := 1, [624].log_data[6].valid := 1, [624].log_data[7].valid := 1, [624].log_data[8].valid := 1, [624].log_data[9].valid := 1, [624].log_data[10].valid := 1, [624].log_data[11].valid := 1, [624].log_data[12].valid := 1, [624].log_data[13].valid := 1, [624].log_data[14].valid := 1, [624].log_data[15].valid := 1,
        [624].log_data[16].valid := 1, [624].log_data[17].valid := 1, [624].log_data[18].valid := 1, [624].log_data[19].valid := 1, [624].time.Year := 2023, [624].time.Month := 1, [624].time.Day := 11, [624].time.Hour := 20, [624].time.Minute := 24, [624].time.Second := 59, [625].log_data[0].min := 1.0, [625].log_data[0].max := 1.0, [625].log_data[0].total := 300.0, [625].log_data[0].time := 300.0, [625].log_data[0].minminute := 25, [625].log_data[0].maxminute := 25, [625].log_data[0].valid := 1, [625].log_data[1].valid := 1, [625].log_data[2].valid := 1, [625].log_data[3].valid := 1, [625].log_data[4].valid := 1, [625].log_data[5].valid := 1, [625].log_data[6].valid := 1, [625].log_data[7].valid := 1, [625].log_data[8].valid := 1, [625].log_data[9].valid := 1, [625].log_data[10].valid := 1, [625].log_data[11].valid := 1, [625].log_data[12].valid := 1, [625].log_data[13].valid := 1, [625].log_data[14].valid := 1, [625].log_data[15].valid := 1, [625].log_data[16].valid := 1, [625].log_data[17].valid := 1, [625].log_data[18].valid := 1, [625].log_data[19].valid := 1, [625].time.Year := 2023, [625].time.Month := 1, [625].time.Day := 11, [625].time.Hour := 20, [625].time.Minute := 29, [625].time.Second := 59, [626].log_data[0].min := 1.0, [626].log_data[0].max := 1.0, [626].log_data[0].total := 300.0, [626].log_data[0].time := 300.0, [626].log_data[0].minminute := 30, [626].log_data[0].maxminute := 30, [626].log_data[0].valid := 1, [626].log_data[1].valid := 1, [626].log_data[2].valid := 1, [626].log_data[3].valid := 1, [626].log_data[4].valid := 1, [626].log_data[5].valid := 1, [626].log_data[6].valid := 1, [626].log_data[7].valid := 1, [626].log_data[8].valid := 1, [626].log_data[9].valid := 1, [626].log_data[10].valid := 1, [626].log_data[11].valid := 1,
        [626].log_data[12].valid := 1, [626].log_data[13].valid := 1, [626].log_data[14].valid := 1, [626].log_data[15].valid := 1, [626].log_data[16].valid := 1, [626].log_data[17].valid := 1, [626].log_data[18].valid := 1, [626].log_data[19].valid := 1, [626].time.Year := 2023, [626].time.Month := 1, [626].time.Day := 11, [626].time.Hour := 20, [626].time.Minute := 34, [626].time.Second := 59, [627].log_data[0].min := 1.0, [627].log_data[0].max := 1.0, [627].log_data[0].total := 300.0, [627].log_data[0].time := 300.0, [627].log_data[0].minminute := 35, [627].log_data[0].maxminute := 35, [627].log_data[0].valid := 1, [627].log_data[1].valid := 1, [627].log_data[2].valid := 1, [627].log_data[3].valid := 1, [627].log_data[4].valid := 1, [627].log_data[5].valid := 1, [627].log_data[6].valid := 1, [627].log_data[7].valid := 1, [627].log_data[8].valid := 1, [627].log_data[9].valid := 1, [627].log_data[10].valid := 1, [627].log_data[11].valid := 1, [627].log_data[12].valid := 1, [627].log_data[13].valid := 1, [627].log_data[14].valid := 1, [627].log_data[15].valid := 1, [627].log_data[16].valid := 1, [627].log_data[17].valid := 1, [627].log_data[18].valid := 1, [627].log_data[19].valid := 1, [627].time.Year := 2023, [627].time.Month := 1, [627].time.Day := 11, [627].time.Hour := 20, [627].time.Minute := 39, [627].time.Second := 59, [628].log_data[0].min := 1.0, [628].log_data[0].max := 1.0, [628].log_data[0].total := 300.0, [628].log_data[0].time := 300.0, [628].log_data[0].minminute := 40, [628].log_data[0].maxminute := 40, [628].log_data[0].valid := 1, [628].log_data[1].valid := 1, [628].log_data[2].valid := 1, [628].log_data[3].valid := 1, [628].log_data[4].valid := 1, [628].log_data[5].valid := 1, [628].log_data[6].valid := 1, [628].log_data[7].valid := 1,
        [628].log_data[8].valid := 1, [628].log_data[9].valid := 1, [628].log_data[10].valid := 1, [628].log_data[11].valid := 1, [628].log_data[12].valid := 1, [628].log_data[13].valid := 1, [628].log_data[14].valid := 1, [628].log_data[15].valid := 1, [628].log_data[16].valid := 1, [628].log_data[17].valid := 1, [628].log_data[18].valid := 1, [628].log_data[19].valid := 1, [628].time.Year := 2023, [628].time.Month := 1, [628].time.Day := 11, [628].time.Hour := 20, [628].time.Minute := 44, [628].time.Second := 59, [629].log_data[0].min := 1.0, [629].log_data[0].max := 1.0, [629].log_data[0].total := 300.0, [629].log_data[0].time := 300.0, [629].log_data[0].minminute := 45, [629].log_data[0].maxminute := 45, [629].log_data[0].valid := 1, [629].log_data[1].valid := 1, [629].log_data[2].valid := 1, [629].log_data[3].valid := 1, [629].log_data[4].valid := 1, [629].log_data[5].valid := 1, [629].log_data[6].valid := 1, [629].log_data[7].valid := 1, [629].log_data[8].valid := 1, [629].log_data[9].valid := 1, [629].log_data[10].valid := 1, [629].log_data[11].valid := 1, [629].log_data[12].valid := 1, [629].log_data[13].valid := 1, [629].log_data[14].valid := 1, [629].log_data[15].valid := 1, [629].log_data[16].valid := 1, [629].log_data[17].valid := 1, [629].log_data[18].valid := 1, [629].log_data[19].valid := 1, [629].time.Year := 2023, [629].time.Month := 1, [629].time.Day := 11, [629].time.Hour := 20, [629].time.Minute := 49, [629].time.Second := 59, [630].log_data[0].min := 1.0, [630].log_data[0].max := 1.0, [630].log_data[0].total := 300.0, [630].log_data[0].time := 300.0, [630].log_data[0].minminute := 50, [630].log_data[0].maxminute := 50, [630].log_data[0].valid := 1, [630].log_data[1].valid := 1, [630].log_data[2].valid := 1, [630].log_data[3].valid := 1,
        [630].log_data[4].valid := 1, [630].log_data[5].valid := 1, [630].log_data[6].valid := 1, [630].log_data[7].valid := 1, [630].log_data[8].valid := 1, [630].log_data[9].valid := 1, [630].log_data[10].valid := 1, [630].log_data[11].valid := 1, [630].log_data[12].valid := 1, [630].log_data[13].valid := 1, [630].log_data[14].valid := 1, [630].log_data[15].valid := 1, [630].log_data[16].valid := 1, [630].log_data[17].valid := 1, [630].log_data[18].valid := 1, [630].log_data[19].valid := 1, [630].time.Year := 2023, [630].time.Month := 1, [630].time.Day := 11, [630].time.Hour := 20, [630].time.Minute := 54, [630].time.Second := 59, [631].log_data[0].min := 1.0, [631].log_data[0].max := 1.0, [631].log_data[0].total := 300.0, [631].log_data[0].time := 300.0, [631].log_data[0].minminute := 55, [631].log_data[0].maxminute := 55, [631].log_data[0].valid := 1, [631].log_data[1].valid := 1, [631].log_data[2].valid := 1, [631].log_data[3].valid := 1, [631].log_data[4].valid := 1, [631].log_data[5].valid := 1, [631].log_data[6].valid := 1, [631].log_data[7].valid := 1, [631].log_data[8].valid := 1, [631].log_data[9].valid := 1, [631].log_data[10].valid := 1, [631].log_data[11].valid := 1, [631].log_data[12].valid := 1, [631].log_data[13].valid := 1, [631].log_data[14].valid := 1, [631].log_data[15].valid := 1, [631].log_data[16].valid := 1, [631].log_data[17].valid := 1, [631].log_data[18].valid := 1, [631].log_data[19].valid := 1, [631].time.Year := 2023, [631].time.Month := 1, [631].time.Day := 11, [631].time.Hour := 20, [631].time.Minute := 59, [631].time.Second := 59, [632].log_data[0].min := 1.0, [632].log_data[0].max := 1.0, [632].log_data[0].total := 300.0, [632].log_data[0].time := 300.0, [632].log_data[0].valid := 1, [632].log_data[1].valid := 1,
        [632].log_data[2].valid := 1, [632].log_data[3].valid := 1, [632].log_data[4].valid := 1, [632].log_data[5].valid := 1, [632].log_data[6].valid := 1, [632].log_data[7].valid := 1, [632].log_data[8].valid := 1, [632].log_data[9].valid := 1, [632].log_data[10].valid := 1, [632].log_data[11].valid := 1, [632].log_data[12].valid := 1, [632].log_data[13].valid := 1, [632].log_data[14].valid := 1, [632].log_data[15].valid := 1, [632].log_data[16].valid := 1, [632].log_data[17].valid := 1, [632].log_data[18].valid := 1, [632].log_data[19].valid := 1, [632].time.Year := 2023, [632].time.Month := 1, [632].time.Day := 11, [632].time.Hour := 21, [632].time.Minute := 4, [632].time.Second := 59, [633].log_data[0].min := 1.0, [633].log_data[0].max := 1.0, [633].log_data[0].total := 300.0, [633].log_data[0].time := 300.0, [633].log_data[0].minminute := 5, [633].log_data[0].maxminute := 5, [633].log_data[0].valid := 1, [633].log_data[1].valid := 1, [633].log_data[2].valid := 1, [633].log_data[3].valid := 1, [633].log_data[4].valid := 1, [633].log_data[5].valid := 1, [633].log_data[6].valid := 1, [633].log_data[7].valid := 1, [633].log_data[8].valid := 1, [633].log_data[9].valid := 1, [633].log_data[10].valid := 1, [633].log_data[11].valid := 1, [633].log_data[12].valid := 1, [633].log_data[13].valid := 1, [633].log_data[14].valid := 1, [633].log_data[15].valid := 1, [633].log_data[16].valid := 1, [633].log_data[17].valid := 1, [633].log_data[18].valid := 1, [633].log_data[19].valid := 1, [633].time.Year := 2023, [633].time.Month := 1, [633].time.Day := 11, [633].time.Hour := 21, [633].time.Minute := 9, [633].time.Second := 59, [634].log_data[0].min := 1.0, [634].log_data[0].max := 1.0, [634].log_data[0].total := 300.0, [634].log_data[0].time := 300.0,
        [634].log_data[0].minminute := 10, [634].log_data[0].maxminute := 10, [634].log_data[0].valid := 1, [634].log_data[1].valid := 1, [634].log_data[2].valid := 1, [634].log_data[3].valid := 1, [634].log_data[4].valid := 1, [634].log_data[5].valid := 1, [634].log_data[6].valid := 1, [634].log_data[7].valid := 1, [634].log_data[8].valid := 1, [634].log_data[9].valid := 1, [634].log_data[10].valid := 1, [634].log_data[11].valid := 1, [634].log_data[12].valid := 1, [634].log_data[13].valid := 1, [634].log_data[14].valid := 1, [634].log_data[15].valid := 1, [634].log_data[16].valid := 1, [634].log_data[17].valid := 1, [634].log_data[18].valid := 1, [634].log_data[19].valid := 1, [634].time.Year := 2023, [634].time.Month := 1, [634].time.Day := 11, [634].time.Hour := 21, [634].time.Minute := 14, [634].time.Second := 59, [635].log_data[0].min := 1.0, [635].log_data[0].max := 1.0, [635].log_data[0].total := 300.0, [635].log_data[0].time := 300.0, [635].log_data[0].minminute := 15, [635].log_data[0].maxminute := 15, [635].log_data[0].valid := 1, [635].log_data[1].valid := 1, [635].log_data[2].valid := 1, [635].log_data[3].valid := 1, [635].log_data[4].valid := 1, [635].log_data[5].valid := 1, [635].log_data[6].valid := 1, [635].log_data[7].valid := 1, [635].log_data[8].valid := 1, [635].log_data[9].valid := 1, [635].log_data[10].valid := 1, [635].log_data[11].valid := 1, [635].log_data[12].valid := 1, [635].log_data[13].valid := 1, [635].log_data[14].valid := 1, [635].log_data[15].valid := 1, [635].log_data[16].valid := 1, [635].log_data[17].valid := 1, [635].log_data[18].valid := 1, [635].log_data[19].valid := 1, [635].time.Year := 2023, [635].time.Month := 1, [635].time.Day := 11, [635].time.Hour := 21, [635].time.Minute := 19, [635].time.Second := 59,
        [636].log_data[0].min := 1.0, [636].log_data[0].max := 1.0, [636].log_data[0].total := 300.0, [636].log_data[0].time := 300.0, [636].log_data[0].minminute := 20, [636].log_data[0].maxminute := 20, [636].log_data[0].valid := 1, [636].log_data[1].valid := 1, [636].log_data[2].valid := 1, [636].log_data[3].valid := 1, [636].log_data[4].valid := 1, [636].log_data[5].valid := 1, [636].log_data[6].valid := 1, [636].log_data[7].valid := 1, [636].log_data[8].valid := 1, [636].log_data[9].valid := 1, [636].log_data[10].valid := 1, [636].log_data[11].valid := 1, [636].log_data[12].valid := 1, [636].log_data[13].valid := 1, [636].log_data[14].valid := 1, [636].log_data[15].valid := 1, [636].log_data[16].valid := 1, [636].log_data[17].valid := 1, [636].log_data[18].valid := 1, [636].log_data[19].valid := 1, [636].time.Year := 2023, [636].time.Month := 1, [636].time.Day := 11, [636].time.Hour := 21, [636].time.Minute := 24, [636].time.Second := 59, [637].log_data[0].min := 1.0, [637].log_data[0].max := 1.0, [637].log_data[0].total := 300.0, [637].log_data[0].time := 300.0, [637].log_data[0].minminute := 25, [637].log_data[0].maxminute := 25, [637].log_data[0].valid := 1, [637].log_data[1].valid := 1, [637].log_data[2].valid := 1, [637].log_data[3].valid := 1, [637].log_data[4].valid := 1, [637].log_data[5].valid := 1, [637].log_data[6].valid := 1, [637].log_data[7].valid := 1, [637].log_data[8].valid := 1, [637].log_data[9].valid := 1, [637].log_data[10].valid := 1, [637].log_data[11].valid := 1, [637].log_data[12].valid := 1, [637].log_data[13].valid := 1, [637].log_data[14].valid := 1, [637].log_data[15].valid := 1, [637].log_data[16].valid := 1, [637].log_data[17].valid := 1, [637].log_data[18].valid := 1, [637].log_data[19].valid := 1, [637].time.Year := 2023, [637].time.Month := 1,
        [637].time.Day := 11, [637].time.Hour := 21, [637].time.Minute := 29, [637].time.Second := 59, [638].log_data[0].min := 1.0, [638].log_data[0].max := 1.0, [638].log_data[0].total := 300.0, [638].log_data[0].time := 300.0, [638].log_data[0].minminute := 30, [638].log_data[0].maxminute := 30, [638].log_data[0].valid := 1, [638].log_data[1].valid := 1, [638].log_data[2].valid := 1, [638].log_data[3].valid := 1, [638].log_data[4].valid := 1, [638].log_data[5].valid := 1, [638].log_data[6].valid := 1, [638].log_data[7].valid := 1, [638].log_data[8].valid := 1, [638].log_data[9].valid := 1, [638].log_data[10].valid := 1, [638].log_data[11].valid := 1, [638].log_data[12].valid := 1, [638].log_data[13].valid := 1, [638].log_data[14].valid := 1, [638].log_data[15].valid := 1, [638].log_data[16].valid := 1, [638].log_data[17].valid := 1, [638].log_data[18].valid := 1, [638].log_data[19].valid := 1, [638].time.Year := 2023, [638].time.Month := 1, [638].time.Day := 11, [638].time.Hour := 21, [638].time.Minute := 34, [638].time.Second := 59, [639].log_data[0].min := 1.0, [639].log_data[0].max := 1.0, [639].log_data[0].total := 300.0, [639].log_data[0].time := 300.0, [639].log_data[0].minminute := 35, [639].log_data[0].maxminute := 35, [639].log_data[0].valid := 1, [639].log_data[1].valid := 1, [639].log_data[2].valid := 1, [639].log_data[3].valid := 1, [639].log_data[4].valid := 1, [639].log_data[5].valid := 1, [639].log_data[6].valid := 1, [639].log_data[7].valid := 1, [639].log_data[8].valid := 1, [639].log_data[9].valid := 1, [639].log_data[10].valid := 1, [639].log_data[11].valid := 1, [639].log_data[12].valid := 1, [639].log_data[13].valid := 1, [639].log_data[14].valid := 1, [639].log_data[15].valid := 1, [639].log_data[16].valid := 1, [639].log_data[17].valid := 1,
        [639].log_data[18].valid := 1, [639].log_data[19].valid := 1, [639].time.Year := 2023, [639].time.Month := 1, [639].time.Day := 11, [639].time.Hour := 21, [639].time.Minute := 39, [639].time.Second := 59, [640].log_data[0].min := 1.0, [640].log_data[0].max := 1.0, [640].log_data[0].total := 300.0, [640].log_data[0].time := 300.0, [640].log_data[0].minminute := 40, [640].log_data[0].maxminute := 40, [640].log_data[0].valid := 1, [640].log_data[1].valid := 1, [640].log_data[2].valid := 1, [640].log_data[3].valid := 1, [640].log_data[4].valid := 1, [640].log_data[5].valid := 1, [640].log_data[6].valid := 1, [640].log_data[7].valid := 1, [640].log_data[8].valid := 1, [640].log_data[9].valid := 1, [640].log_data[10].valid := 1, [640].log_data[11].valid := 1, [640].log_data[12].valid := 1, [640].log_data[13].valid := 1, [640].log_data[14].valid := 1, [640].log_data[15].valid := 1, [640].log_data[16].valid := 1, [640].log_data[17].valid := 1, [640].log_data[18].valid := 1, [640].log_data[19].valid := 1, [640].time.Year := 2023, [640].time.Month := 1, [640].time.Day := 11, [640].time.Hour := 21, [640].time.Minute := 44, [640].time.Second := 59, [641].log_data[0].min := 1.0, [641].log_data[0].max := 1.0, [641].log_data[0].total := 300.0, [641].log_data[0].time := 300.0, [641].log_data[0].minminute := 45, [641].log_data[0].maxminute := 45, [641].log_data[0].valid := 1, [641].log_data[1].valid := 1, [641].log_data[2].valid := 1, [641].log_data[3].valid := 1, [641].log_data[4].valid := 1, [641].log_data[5].valid := 1, [641].log_data[6].valid := 1, [641].log_data[7].valid := 1, [641].log_data[8].valid := 1, [641].log_data[9].valid := 1, [641].log_data[10].valid := 1, [641].log_data[11].valid := 1, [641].log_data[12].valid := 1, [641].log_data[13].valid := 1,
        [641].log_data[14].valid := 1, [641].log_data[15].valid := 1, [641].log_data[16].valid := 1, [641].log_data[17].valid := 1, [641].log_data[18].valid := 1, [641].log_data[19].valid := 1, [641].time.Year := 2023, [641].time.Month := 1, [641].time.Day := 11, [641].time.Hour := 21, [641].time.Minute := 49, [641].time.Second := 59, [642].log_data[0].min := 1.0, [642].log_data[0].max := 1.0, [642].log_data[0].total := 300.0, [642].log_data[0].time := 300.0, [642].log_data[0].minminute := 50, [642].log_data[0].maxminute := 50, [642].log_data[0].valid := 1, [642].log_data[1].valid := 1, [642].log_data[2].valid := 1, [642].log_data[3].valid := 1, [642].log_data[4].valid := 1, [642].log_data[5].valid := 1, [642].log_data[6].valid := 1, [642].log_data[7].valid := 1, [642].log_data[8].valid := 1, [642].log_data[9].valid := 1, [642].log_data[10].valid := 1, [642].log_data[11].valid := 1, [642].log_data[12].valid := 1, [642].log_data[13].valid := 1, [642].log_data[14].valid := 1, [642].log_data[15].valid := 1, [642].log_data[16].valid := 1, [642].log_data[17].valid := 1, [642].log_data[18].valid := 1, [642].log_data[19].valid := 1, [642].time.Year := 2023, [642].time.Month := 1, [642].time.Day := 11, [642].time.Hour := 21, [642].time.Minute := 54, [642].time.Second := 59, [643].log_data[0].min := 1.0, [643].log_data[0].max := 1.0, [643].log_data[0].total := 300.0, [643].log_data[0].time := 300.0, [643].log_data[0].minminute := 55, [643].log_data[0].maxminute := 55, [643].log_data[0].valid := 1, [643].log_data[1].valid := 1, [643].log_data[2].valid := 1, [643].log_data[3].valid := 1, [643].log_data[4].valid := 1, [643].log_data[5].valid := 1, [643].log_data[6].valid := 1, [643].log_data[7].valid := 1, [643].log_data[8].valid := 1, [643].log_data[9].valid := 1,
        [643].log_data[10].valid := 1, [643].log_data[11].valid := 1, [643].log_data[12].valid := 1, [643].log_data[13].valid := 1, [643].log_data[14].valid := 1, [643].log_data[15].valid := 1, [643].log_data[16].valid := 1, [643].log_data[17].valid := 1, [643].log_data[18].valid := 1, [643].log_data[19].valid := 1, [643].time.Year := 2023, [643].time.Month := 1, [643].time.Day := 11, [643].time.Hour := 21, [643].time.Minute := 59, [643].time.Second := 59, [644].log_data[0].min := 1.0, [644].log_data[0].max := 1.0, [644].log_data[0].total := 300.0, [644].log_data[0].time := 300.0, [644].log_data[0].valid := 1, [644].log_data[1].valid := 1, [644].log_data[2].valid := 1, [644].log_data[3].valid := 1, [644].log_data[4].valid := 1, [644].log_data[5].valid := 1, [644].log_data[6].valid := 1, [644].log_data[7].valid := 1, [644].log_data[8].valid := 1, [644].log_data[9].valid := 1, [644].log_data[10].valid := 1, [644].log_data[11].valid := 1, [644].log_data[12].valid := 1, [644].log_data[13].valid := 1, [644].log_data[14].valid := 1, [644].log_data[15].valid := 1, [644].log_data[16].valid := 1, [644].log_data[17].valid := 1, [644].log_data[18].valid := 1, [644].log_data[19].valid := 1, [644].time.Year := 2023, [644].time.Month := 1, [644].time.Day := 11, [644].time.Hour := 22, [644].time.Minute := 4, [644].time.Second := 59, [645].log_data[0].min := 1.0, [645].log_data[0].max := 1.0, [645].log_data[0].total := 300.0, [645].log_data[0].time := 300.0, [645].log_data[0].minminute := 5, [645].log_data[0].maxminute := 5, [645].log_data[0].valid := 1, [645].log_data[1].valid := 1, [645].log_data[2].valid := 1, [645].log_data[3].valid := 1, [645].log_data[4].valid := 1, [645].log_data[5].valid := 1, [645].log_data[6].valid := 1, [645].log_data[7].valid := 1,
        [645].log_data[8].valid := 1, [645].log_data[9].valid := 1, [645].log_data[10].valid := 1, [645].log_data[11].valid := 1, [645].log_data[12].valid := 1, [645].log_data[13].valid := 1, [645].log_data[14].valid := 1, [645].log_data[15].valid := 1, [645].log_data[16].valid := 1, [645].log_data[17].valid := 1, [645].log_data[18].valid := 1, [645].log_data[19].valid := 1, [645].time.Year := 2023, [645].time.Month := 1, [645].time.Day := 11, [645].time.Hour := 22, [645].time.Minute := 9, [645].time.Second := 59, [646].log_data[0].min := 1.0, [646].log_data[0].max := 1.0, [646].log_data[0].total := 300.0, [646].log_data[0].time := 300.0, [646].log_data[0].minminute := 10, [646].log_data[0].maxminute := 10, [646].log_data[0].valid := 1, [646].log_data[1].valid := 1, [646].log_data[2].valid := 1, [646].log_data[3].valid := 1, [646].log_data[4].valid := 1, [646].log_data[5].valid := 1, [646].log_data[6].valid := 1, [646].log_data[7].valid := 1, [646].log_data[8].valid := 1, [646].log_data[9].valid := 1, [646].log_data[10].valid := 1, [646].log_data[11].valid := 1, [646].log_data[12].valid := 1, [646].log_data[13].valid := 1, [646].log_data[14].valid := 1, [646].log_data[15].valid := 1, [646].log_data[16].valid := 1, [646].log_data[17].valid := 1, [646].log_data[18].valid := 1, [646].log_data[19].valid := 1, [646].time.Year := 2023, [646].time.Month := 1, [646].time.Day := 11, [646].time.Hour := 22, [646].time.Minute := 14, [646].time.Second := 59, [647].log_data[0].min := 1.0, [647].log_data[0].max := 1.0, [647].log_data[0].total := 300.0, [647].log_data[0].time := 300.0, [647].log_data[0].minminute := 15, [647].log_data[0].maxminute := 15, [647].log_data[0].valid := 1, [647].log_data[1].valid := 1, [647].log_data[2].valid := 1, [647].log_data[3].valid := 1,
        [647].log_data[4].valid := 1, [647].log_data[5].valid := 1, [647].log_data[6].valid := 1, [647].log_data[7].valid := 1, [647].log_data[8].valid := 1, [647].log_data[9].valid := 1, [647].log_data[10].valid := 1, [647].log_data[11].valid := 1, [647].log_data[12].valid := 1, [647].log_data[13].valid := 1, [647].log_data[14].valid := 1, [647].log_data[15].valid := 1, [647].log_data[16].valid := 1, [647].log_data[17].valid := 1, [647].log_data[18].valid := 1, [647].log_data[19].valid := 1, [647].time.Year := 2023, [647].time.Month := 1, [647].time.Day := 11, [647].time.Hour := 22, [647].time.Minute := 19, [647].time.Second := 59, [648].log_data[0].min := 1.0, [648].log_data[0].max := 1.0, [648].log_data[0].total := 300.0, [648].log_data[0].time := 300.0, [648].log_data[0].minminute := 20, [648].log_data[0].maxminute := 20, [648].log_data[0].valid := 1, [648].log_data[1].valid := 1, [648].log_data[2].valid := 1, [648].log_data[3].valid := 1, [648].log_data[4].valid := 1, [648].log_data[5].valid := 1, [648].log_data[6].valid := 1, [648].log_data[7].valid := 1, [648].log_data[8].valid := 1, [648].log_data[9].valid := 1, [648].log_data[10].valid := 1, [648].log_data[11].valid := 1, [648].log_data[12].valid := 1, [648].log_data[13].valid := 1, [648].log_data[14].valid := 1, [648].log_data[15].valid := 1, [648].log_data[16].valid := 1, [648].log_data[17].valid := 1, [648].log_data[18].valid := 1, [648].log_data[19].valid := 1, [648].time.Year := 2023, [648].time.Month := 1, [648].time.Day := 11, [648].time.Hour := 22, [648].time.Minute := 24, [648].time.Second := 59, [649].log_data[0].min := 1.0, [649].log_data[0].max := 1.0, [649].log_data[0].total := 300.0, [649].log_data[0].time := 300.0, [649].log_data[0].minminute := 25, [649].log_data[0].maxminute := 25,
        [649].log_data[0].valid := 1, [649].log_data[1].valid := 1, [649].log_data[2].valid := 1, [649].log_data[3].valid := 1, [649].log_data[4].valid := 1, [649].log_data[5].valid := 1, [649].log_data[6].valid := 1, [649].log_data[7].valid := 1, [649].log_data[8].valid := 1, [649].log_data[9].valid := 1, [649].log_data[10].valid := 1, [649].log_data[11].valid := 1, [649].log_data[12].valid := 1, [649].log_data[13].valid := 1, [649].log_data[14].valid := 1, [649].log_data[15].valid := 1, [649].log_data[16].valid := 1, [649].log_data[17].valid := 1, [649].log_data[18].valid := 1, [649].log_data[19].valid := 1, [649].time.Year := 2023, [649].time.Month := 1, [649].time.Day := 11, [649].time.Hour := 22, [649].time.Minute := 29, [649].time.Second := 59, [650].log_data[0].min := 1.0, [650].log_data[0].max := 1.0, [650].log_data[0].total := 300.0, [650].log_data[0].time := 300.0, [650].log_data[0].minminute := 30, [650].log_data[0].maxminute := 30, [650].log_data[0].valid := 1, [650].log_data[1].valid := 1, [650].log_data[2].valid := 1, [650].log_data[3].valid := 1, [650].log_data[4].valid := 1, [650].log_data[5].valid := 1, [650].log_data[6].valid := 1, [650].log_data[7].valid := 1, [650].log_data[8].valid := 1, [650].log_data[9].valid := 1, [650].log_data[10].valid := 1, [650].log_data[11].valid := 1, [650].log_data[12].valid := 1, [650].log_data[13].valid := 1, [650].log_data[14].valid := 1, [650].log_data[15].valid := 1, [650].log_data[16].valid := 1, [650].log_data[17].valid := 1, [650].log_data[18].valid := 1, [650].log_data[19].valid := 1, [650].time.Year := 2023, [650].time.Month := 1, [650].time.Day := 11, [650].time.Hour := 22, [650].time.Minute := 34, [650].time.Second := 59, [651].log_data[0].min := 1.0, [651].log_data[0].max := 1.0,
        [651].log_data[0].total := 300.0, [651].log_data[0].time := 300.0, [651].log_data[0].minminute := 35, [651].log_data[0].maxminute := 35, [651].log_data[0].valid := 1, [651].log_data[1].valid := 1, [651].log_data[2].valid := 1, [651].log_data[3].valid := 1, [651].log_data[4].valid := 1, [651].log_data[5].valid := 1, [651].log_data[6].valid := 1, [651].log_data[7].valid := 1, [651].log_data[8].valid := 1, [651].log_data[9].valid := 1, [651].log_data[10].valid := 1, [651].log_data[11].valid := 1, [651].log_data[12].valid := 1, [651].log_data[13].valid := 1, [651].log_data[14].valid := 1, [651].log_data[15].valid := 1, [651].log_data[16].valid := 1, [651].log_data[17].valid := 1, [651].log_data[18].valid := 1, [651].log_data[19].valid := 1, [651].time.Year := 2023, [651].time.Month := 1, [651].time.Day := 11, [651].time.Hour := 22, [651].time.Minute := 39, [651].time.Second := 59, [652].log_data[0].min := 1.0, [652].log_data[0].max := 1.0, [652].log_data[0].total := 300.0, [652].log_data[0].time := 300.0, [652].log_data[0].minminute := 40, [652].log_data[0].maxminute := 40, [652].log_data[0].valid := 1, [652].log_data[1].valid := 1, [652].log_data[2].valid := 1, [652].log_data[3].valid := 1, [652].log_data[4].valid := 1, [652].log_data[5].valid := 1, [652].log_data[6].valid := 1, [652].log_data[7].valid := 1, [652].log_data[8].valid := 1, [652].log_data[9].valid := 1, [652].log_data[10].valid := 1, [652].log_data[11].valid := 1, [652].log_data[12].valid := 1, [652].log_data[13].valid := 1, [652].log_data[14].valid := 1, [652].log_data[15].valid := 1, [652].log_data[16].valid := 1, [652].log_data[17].valid := 1, [652].log_data[18].valid := 1, [652].log_data[19].valid := 1, [652].time.Year := 2023, [652].time.Month := 1, [652].time.Day := 11, [652].time.Hour := 22,
        [652].time.Minute := 44, [652].time.Second := 59, [653].log_data[0].min := 1.0, [653].log_data[0].max := 1.0, [653].log_data[0].total := 300.0, [653].log_data[0].time := 300.0, [653].log_data[0].minminute := 45, [653].log_data[0].maxminute := 45, [653].log_data[0].valid := 1, [653].log_data[1].valid := 1, [653].log_data[2].valid := 1, [653].log_data[3].valid := 1, [653].log_data[4].valid := 1, [653].log_data[5].valid := 1, [653].log_data[6].valid := 1, [653].log_data[7].valid := 1, [653].log_data[8].valid := 1, [653].log_data[9].valid := 1, [653].log_data[10].valid := 1, [653].log_data[11].valid := 1, [653].log_data[12].valid := 1, [653].log_data[13].valid := 1, [653].log_data[14].valid := 1, [653].log_data[15].valid := 1, [653].log_data[16].valid := 1, [653].log_data[17].valid := 1, [653].log_data[18].valid := 1, [653].log_data[19].valid := 1, [653].time.Year := 2023, [653].time.Month := 1, [653].time.Day := 11, [653].time.Hour := 22, [653].time.Minute := 49, [653].time.Second := 59, [654].log_data[0].min := 1.0, [654].log_data[0].max := 1.0, [654].log_data[0].total := 300.0, [654].log_data[0].time := 300.0, [654].log_data[0].minminute := 50, [654].log_data[0].maxminute := 50, [654].log_data[0].valid := 1, [654].log_data[1].valid := 1, [654].log_data[2].valid := 1, [654].log_data[3].valid := 1, [654].log_data[4].valid := 1, [654].log_data[5].valid := 1, [654].log_data[6].valid := 1, [654].log_data[7].valid := 1, [654].log_data[8].valid := 1, [654].log_data[9].valid := 1, [654].log_data[10].valid := 1, [654].log_data[11].valid := 1, [654].log_data[12].valid := 1, [654].log_data[13].valid := 1, [654].log_data[14].valid := 1, [654].log_data[15].valid := 1, [654].log_data[16].valid := 1, [654].log_data[17].valid := 1, [654].log_data[18].valid := 1, [654].log_data[19].valid := 1,
        [654].time.Year := 2023, [654].time.Month := 1, [654].time.Day := 11, [654].time.Hour := 22, [654].time.Minute := 54, [654].time.Second := 59, [655].log_data[0].min := 1.0, [655].log_data[0].max := 1.0, [655].log_data[0].total := 300.0, [655].log_data[0].time := 300.0, [655].log_data[0].minminute := 55, [655].log_data[0].maxminute := 55, [655].log_data[0].valid := 1, [655].log_data[1].valid := 1, [655].log_data[2].valid := 1, [655].log_data[3].valid := 1, [655].log_data[4].valid := 1, [655].log_data[5].valid := 1, [655].log_data[6].valid := 1, [655].log_data[7].valid := 1, [655].log_data[8].valid := 1, [655].log_data[9].valid := 1, [655].log_data[10].valid := 1, [655].log_data[11].valid := 1, [655].log_data[12].valid := 1, [655].log_data[13].valid := 1, [655].log_data[14].valid := 1, [655].log_data[15].valid := 1, [655].log_data[16].valid := 1, [655].log_data[17].valid := 1, [655].log_data[18].valid := 1, [655].log_data[19].valid := 1, [655].time.Year := 2023, [655].time.Month := 1, [655].time.Day := 11, [655].time.Hour := 22, [655].time.Minute := 59, [655].time.Second := 59, [656].log_data[0].min := 1.0, [656].log_data[0].max := 1.0, [656].log_data[0].total := 300.0, [656].log_data[0].time := 300.0, [656].log_data[0].valid := 1, [656].log_data[1].valid := 1, [656].log_data[2].valid := 1, [656].log_data[3].valid := 1, [656].log_data[4].valid := 1, [656].log_data[5].valid := 1, [656].log_data[6].valid := 1, [656].log_data[7].valid := 1, [656].log_data[8].valid := 1, [656].log_data[9].valid := 1, [656].log_data[10].valid := 1, [656].log_data[11].valid := 1, [656].log_data[12].valid := 1, [656].log_data[13].valid := 1, [656].log_data[14].valid := 1, [656].log_data[15].valid := 1, [656].log_data[16].valid := 1, [656].log_data[17].valid := 1,
        [656].log_data[18].valid := 1, [656].log_data[19].valid := 1, [656].time.Year := 2023, [656].time.Month := 1, [656].time.Day := 11, [656].time.Hour := 23, [656].time.Minute := 4, [656].time.Second := 59, [657].log_data[0].min := 1.0, [657].log_data[0].max := 1.0, [657].log_data[0].total := 300.0, [657].log_data[0].time := 300.0, [657].log_data[0].minminute := 5, [657].log_data[0].maxminute := 5, [657].log_data[0].valid := 1, [657].log_data[1].valid := 1, [657].log_data[2].valid := 1, [657].log_data[3].valid := 1, [657].log_data[4].valid := 1, [657].log_data[5].valid := 1, [657].log_data[6].valid := 1, [657].log_data[7].valid := 1, [657].log_data[8].valid := 1, [657].log_data[9].valid := 1, [657].log_data[10].valid := 1, [657].log_data[11].valid := 1, [657].log_data[12].valid := 1, [657].log_data[13].valid := 1, [657].log_data[14].valid := 1, [657].log_data[15].valid := 1, [657].log_data[16].valid := 1, [657].log_data[17].valid := 1, [657].log_data[18].valid := 1, [657].log_data[19].valid := 1, [657].time.Year := 2023, [657].time.Month := 1, [657].time.Day := 11, [657].time.Hour := 23, [657].time.Minute := 9, [657].time.Second := 59, [658].log_data[0].min := 1.0, [658].log_data[0].max := 1.0, [658].log_data[0].total := 300.0, [658].log_data[0].time := 300.0, [658].log_data[0].minminute := 10, [658].log_data[0].maxminute := 10, [658].log_data[0].valid := 1, [658].log_data[1].valid := 1, [658].log_data[2].valid := 1, [658].log_data[3].valid := 1, [658].log_data[4].valid := 1, [658].log_data[5].valid := 1, [658].log_data[6].valid := 1, [658].log_data[7].valid := 1, [658].log_data[8].valid := 1, [658].log_data[9].valid := 1, [658].log_data[10].valid := 1, [658].log_data[11].valid := 1, [658].log_data[12].valid := 1, [658].log_data[13].valid := 1,
        [658].log_data[14].valid := 1, [658].log_data[15].valid := 1, [658].log_data[16].valid := 1, [658].log_data[17].valid := 1, [658].log_data[18].valid := 1, [658].log_data[19].valid := 1, [658].time.Year := 2023, [658].time.Month := 1, [658].time.Day := 11, [658].time.Hour := 23, [658].time.Minute := 14, [658].time.Second := 59, [659].log_data[0].min := 1.0, [659].log_data[0].max := 1.0, [659].log_data[0].total := 300.0, [659].log_data[0].time := 300.0, [659].log_data[0].minminute := 15, [659].log_data[0].maxminute := 15, [659].log_data[0].valid := 1, [659].log_data[1].valid := 1, [659].log_data[2].valid := 1, [659].log_data[3].valid := 1, [659].log_data[4].valid := 1, [659].log_data[5].valid := 1, [659].log_data[6].valid := 1, [659].log_data[7].valid := 1, [659].log_data[8].valid := 1, [659].log_data[9].valid := 1, [659].log_data[10].valid := 1, [659].log_data[11].valid := 1, [659].log_data[12].valid := 1, [659].log_data[13].valid := 1, [659].log_data[14].valid := 1, [659].log_data[15].valid := 1, [659].log_data[16].valid := 1, [659].log_data[17].valid := 1, [659].log_data[18].valid := 1, [659].log_data[19].valid := 1, [659].time.Year := 2023, [659].time.Month := 1, [659].time.Day := 11, [659].time.Hour := 23, [659].time.Minute := 19, [659].time.Second := 59, [660].log_data[0].min := 1.0, [660].log_data[0].max := 1.0, [660].log_data[0].total := 300.0, [660].log_data[0].time := 300.0, [660].log_data[0].minminute := 20, [660].log_data[0].maxminute := 20, [660].log_data[0].valid := 1, [660].log_data[1].valid := 1, [660].log_data[2].valid := 1, [660].log_data[3].valid := 1, [660].log_data[4].valid := 1, [660].log_data[5].valid := 1, [660].log_data[6].valid := 1, [660].log_data[7].valid := 1, [660].log_data[8].valid := 1, [660].log_data[9].valid := 1,
        [660].log_data[10].valid := 1, [660].log_data[11].valid := 1, [660].log_data[12].valid := 1, [660].log_data[13].valid := 1, [660].log_data[14].valid := 1, [660].log_data[15].valid := 1, [660].log_data[16].valid := 1, [660].log_data[17].valid := 1, [660].log_data[18].valid := 1, [660].log_data[19].valid := 1, [660].time.Year := 2023, [660].time.Month := 1, [660].time.Day := 11, [660].time.Hour := 23, [660].time.Minute := 24, [660].time.Second := 59, [661].log_data[0].min := 1.0, [661].log_data[0].max := 1.0, [661].log_data[0].total := 300.0, [661].log_data[0].time := 300.0, [661].log_data[0].minminute := 25, [661].log_data[0].maxminute := 25, [661].log_data[0].valid := 1, [661].log_data[1].valid := 1, [661].log_data[2].valid := 1, [661].log_data[3].valid := 1, [661].log_data[4].valid := 1, [661].log_data[5].valid := 1, [661].log_data[6].valid := 1, [661].log_data[7].valid := 1, [661].log_data[8].valid := 1, [661].log_data[9].valid := 1, [661].log_data[10].valid := 1, [661].log_data[11].valid := 1, [661].log_data[12].valid := 1, [661].log_data[13].valid := 1, [661].log_data[14].valid := 1, [661].log_data[15].valid := 1, [661].log_data[16].valid := 1, [661].log_data[17].valid := 1, [661].log_data[18].valid := 1, [661].log_data[19].valid := 1, [661].time.Year := 2023, [661].time.Month := 1, [661].time.Day := 11, [661].time.Hour := 23, [661].time.Minute := 29, [661].time.Second := 59, [662].log_data[0].min := 1.0, [662].log_data[0].max := 1.0, [662].log_data[0].total := 300.0, [662].log_data[0].time := 300.0, [662].log_data[0].minminute := 30, [662].log_data[0].maxminute := 30, [662].log_data[0].valid := 1, [662].log_data[1].valid := 1, [662].log_data[2].valid := 1, [662].log_data[3].valid := 1, [662].log_data[4].valid := 1, [662].log_data[5].valid := 1,
        [662].log_data[6].valid := 1, [662].log_data[7].valid := 1, [662].log_data[8].valid := 1, [662].log_data[9].valid := 1, [662].log_data[10].valid := 1, [662].log_data[11].valid := 1, [662].log_data[12].valid := 1, [662].log_data[13].valid := 1, [662].log_data[14].valid := 1, [662].log_data[15].valid := 1, [662].log_data[16].valid := 1, [662].log_data[17].valid := 1, [662].log_data[18].valid := 1, [662].log_data[19].valid := 1, [662].time.Year := 2023, [662].time.Month := 1, [662].time.Day := 11, [662].time.Hour := 23, [662].time.Minute := 34, [662].time.Second := 59, [663].log_data[0].min := 1.0, [663].log_data[0].max := 1.0, [663].log_data[0].total := 300.0, [663].log_data[0].time := 300.0, [663].log_data[0].minminute := 35, [663].log_data[0].maxminute := 35, [663].log_data[0].valid := 1, [663].log_data[1].valid := 1, [663].log_data[2].valid := 1, [663].log_data[3].valid := 1, [663].log_data[4].valid := 1, [663].log_data[5].valid := 1, [663].log_data[6].valid := 1, [663].log_data[7].valid := 1, [663].log_data[8].valid := 1, [663].log_data[9].valid := 1, [663].log_data[10].valid := 1, [663].log_data[11].valid := 1, [663].log_data[12].valid := 1, [663].log_data[13].valid := 1, [663].log_data[14].valid := 1, [663].log_data[15].valid := 1, [663].log_data[16].valid := 1, [663].log_data[17].valid := 1, [663].log_data[18].valid := 1, [663].log_data[19].valid := 1, [663].time.Year := 2023, [663].time.Month := 1, [663].time.Day := 11, [663].time.Hour := 23, [663].time.Minute := 39, [663].time.Second := 59, [664].log_data[0].min := 1.0, [664].log_data[0].max := 1.0, [664].log_data[0].total := 300.0, [664].log_data[0].time := 300.0, [664].log_data[0].minminute := 40, [664].log_data[0].maxminute := 40, [664].log_data[0].valid := 1, [664].log_data[1].valid := 1,
        [664].log_data[2].valid := 1, [664].log_data[3].valid := 1, [664].log_data[4].valid := 1, [664].log_data[5].valid := 1, [664].log_data[6].valid := 1, [664].log_data[7].valid := 1, [664].log_data[8].valid := 1, [664].log_data[9].valid := 1, [664].log_data[10].valid := 1, [664].log_data[11].valid := 1, [664].log_data[12].valid := 1, [664].log_data[13].valid := 1, [664].log_data[14].valid := 1, [664].log_data[15].valid := 1, [664].log_data[16].valid := 1, [664].log_data[17].valid := 1, [664].log_data[18].valid := 1, [664].log_data[19].valid := 1, [664].time.Year := 2023, [664].time.Month := 1, [664].time.Day := 11, [664].time.Hour := 23, [664].time.Minute := 44, [664].time.Second := 59, [665].log_data[0].min := 1.0, [665].log_data[0].max := 1.0, [665].log_data[0].total := 300.0, [665].log_data[0].time := 300.0, [665].log_data[0].minminute := 45, [665].log_data[0].maxminute := 45, [665].log_data[0].valid := 1, [665].log_data[1].valid := 1, [665].log_data[2].valid := 1, [665].log_data[3].valid := 1, [665].log_data[4].valid := 1, [665].log_data[5].valid := 1, [665].log_data[6].valid := 1, [665].log_data[7].valid := 1, [665].log_data[8].valid := 1, [665].log_data[9].valid := 1, [665].log_data[10].valid := 1, [665].log_data[11].valid := 1, [665].log_data[12].valid := 1, [665].log_data[13].valid := 1, [665].log_data[14].valid := 1, [665].log_data[15].valid := 1, [665].log_data[16].valid := 1, [665].log_data[17].valid := 1, [665].log_data[18].valid := 1, [665].log_data[19].valid := 1, [665].time.Year := 2023, [665].time.Month := 1, [665].time.Day := 11, [665].time.Hour := 23, [665].time.Minute := 49, [665].time.Second := 59, [666].log_data[0].min := 1.0, [666].log_data[0].max := 1.0, [666].log_data[0].total := 300.0, [666].log_data[0].time := 300.0,
        [666].log_data[0].minminute := 50, [666].log_data[0].maxminute := 50, [666].log_data[0].valid := 1, [666].log_data[1].valid := 1, [666].log_data[2].valid := 1, [666].log_data[3].valid := 1, [666].log_data[4].valid := 1, [666].log_data[5].valid := 1, [666].log_data[6].valid := 1, [666].log_data[7].valid := 1, [666].log_data[8].valid := 1, [666].log_data[9].valid := 1, [666].log_data[10].valid := 1, [666].log_data[11].valid := 1, [666].log_data[12].valid := 1, [666].log_data[13].valid := 1, [666].log_data[14].valid := 1, [666].log_data[15].valid := 1, [666].log_data[16].valid := 1, [666].log_data[17].valid := 1, [666].log_data[18].valid := 1, [666].log_data[19].valid := 1, [666].time.Year := 2023, [666].time.Month := 1, [666].time.Day := 11, [666].time.Hour := 23, [666].time.Minute := 54, [666].time.Second := 59, [667].log_data[0].min := 1.0, [667].log_data[0].max := 1.0, [667].log_data[0].total := 300.0, [667].log_data[0].time := 300.0, [667].log_data[0].minminute := 55, [667].log_data[0].maxminute := 55, [667].log_data[0].valid := 1, [667].log_data[1].valid := 1, [667].log_data[2].valid := 1, [667].log_data[3].valid := 1, [667].log_data[4].valid := 1, [667].log_data[5].valid := 1, [667].log_data[6].valid := 1, [667].log_data[7].valid := 1, [667].log_data[8].valid := 1, [667].log_data[9].valid := 1, [667].log_data[10].valid := 1, [667].log_data[11].valid := 1, [667].log_data[12].valid := 1, [667].log_data[13].valid := 1, [667].log_data[14].valid := 1, [667].log_data[15].valid := 1, [667].log_data[16].valid := 1, [667].log_data[17].valid := 1, [667].log_data[18].valid := 1, [667].log_data[19].valid := 1, [667].time.Year := 2023, [667].time.Month := 1, [667].time.Day := 11, [667].time.Hour := 23, [667].time.Minute := 59, [667].time.Second := 59,
        [668].log_data[0].min := 1.0, [668].log_data[0].max := 1.0, [668].log_data[0].total := 300.0, [668].log_data[0].time := 300.0, [668].log_data[0].valid := 1, [668].log_data[1].valid := 1, [668].log_data[2].valid := 1, [668].log_data[3].valid := 1, [668].log_data[4].valid := 1, [668].log_data[5].valid := 1, [668].log_data[6].valid := 1, [668].log_data[7].valid := 1, [668].log_data[8].valid := 1, [668].log_data[9].valid := 1, [668].log_data[10].valid := 1, [668].log_data[11].valid := 1, [668].log_data[12].valid := 1, [668].log_data[13].valid := 1, [668].log_data[14].valid := 1, [668].log_data[15].valid := 1, [668].log_data[16].valid := 1, [668].log_data[17].valid := 1, [668].log_data[18].valid := 1, [668].log_data[19].valid := 1, [668].time.Year := 2023, [668].time.Month := 1, [668].time.Day := 12, [668].time.Minute := 4, [668].time.Second := 59, [669].log_data[0].min := 1.0, [669].log_data[0].max := 1.0, [669].log_data[0].total := 300.0, [669].log_data[0].time := 300.0, [669].log_data[0].minminute := 5, [669].log_data[0].maxminute := 5, [669].log_data[0].valid := 1, [669].log_data[1].valid := 1, [669].log_data[2].valid := 1, [669].log_data[3].valid := 1, [669].log_data[4].valid := 1, [669].log_data[5].valid := 1, [669].log_data[6].valid := 1, [669].log_data[7].valid := 1, [669].log_data[8].valid := 1, [669].log_data[9].valid := 1, [669].log_data[10].valid := 1, [669].log_data[11].valid := 1, [669].log_data[12].valid := 1, [669].log_data[13].valid := 1, [669].log_data[14].valid := 1, [669].log_data[15].valid := 1, [669].log_data[16].valid := 1, [669].log_data[17].valid := 1, [669].log_data[18].valid := 1, [669].log_data[19].valid := 1, [669].time.Year := 2023, [669].time.Month := 1, [669].time.Day := 12, [669].time.Minute := 9, [669].time.Second := 59,
        [670].log_data[0].min := 1.0, [670].log_data[0].max := 1.0, [670].log_data[0].total := 300.0, [670].log_data[0].time := 300.0, [670].log_data[0].minminute := 10, [670].log_data[0].maxminute := 10, [670].log_data[0].valid := 1, [670].log_data[1].valid := 1, [670].log_data[2].valid := 1, [670].log_data[3].valid := 1, [670].log_data[4].valid := 1, [670].log_data[5].valid := 1, [670].log_data[6].valid := 1, [670].log_data[7].valid := 1, [670].log_data[8].valid := 1, [670].log_data[9].valid := 1, [670].log_data[10].valid := 1, [670].log_data[11].valid := 1, [670].log_data[12].valid := 1, [670].log_data[13].valid := 1, [670].log_data[14].valid := 1, [670].log_data[15].valid := 1, [670].log_data[16].valid := 1, [670].log_data[17].valid := 1, [670].log_data[18].valid := 1, [670].log_data[19].valid := 1, [670].time.Year := 2023, [670].time.Month := 1, [670].time.Day := 12, [670].time.Minute := 14, [670].time.Second := 59, [671].log_data[0].min := 1.0, [671].log_data[0].max := 1.0, [671].log_data[0].total := 300.0, [671].log_data[0].time := 300.0, [671].log_data[0].minminute := 15, [671].log_data[0].maxminute := 15, [671].log_data[0].valid := 1, [671].log_data[1].valid := 1, [671].log_data[2].valid := 1, [671].log_data[3].valid := 1, [671].log_data[4].valid := 1, [671].log_data[5].valid := 1, [671].log_data[6].valid := 1, [671].log_data[7].valid := 1, [671].log_data[8].valid := 1, [671].log_data[9].valid := 1, [671].log_data[10].valid := 1, [671].log_data[11].valid := 1, [671].log_data[12].valid := 1, [671].log_data[13].valid := 1, [671].log_data[14].valid := 1, [671].log_data[15].valid := 1, [671].log_data[16].valid := 1, [671].log_data[17].valid := 1, [671].log_data[18].valid := 1, [671].log_data[19].valid := 1, [671].time.Year := 2023, [671].time.Month := 1, [671].time.Day := 12,
        [671].time.Minute := 19, [671].time.Second := 59, [672].log_data[0].min := 1.0, [672].log_data[0].max := 1.0, [672].log_data[0].total := 300.0, [672].log_data[0].time := 300.0, [672].log_data[0].minminute := 20, [672].log_data[0].maxminute := 20, [672].log_data[0].valid := 1, [672].log_data[1].valid := 1, [672].log_data[2].valid := 1, [672].log_data[3].valid := 1, [672].log_data[4].valid := 1, [672].log_data[5].valid := 1, [672].log_data[6].valid := 1, [672].log_data[7].valid := 1, [672].log_data[8].valid := 1, [672].log_data[9].valid := 1, [672].log_data[10].valid := 1, [672].log_data[11].valid := 1, [672].log_data[12].valid := 1, [672].log_data[13].valid := 1, [672].log_data[14].valid := 1, [672].log_data[15].valid := 1, [672].log_data[16].valid := 1, [672].log_data[17].valid := 1, [672].log_data[18].valid := 1, [672].log_data[19].valid := 1, [672].time.Year := 2023, [672].time.Month := 1, [672].time.Day := 12, [672].time.Minute := 24, [672].time.Second := 59, [673].log_data[0].min := 1.0, [673].log_data[0].max := 1.0, [673].log_data[0].total := 300.0, [673].log_data[0].time := 300.0, [673].log_data[0].minminute := 25, [673].log_data[0].maxminute := 25, [673].log_data[0].valid := 1, [673].log_data[1].valid := 1, [673].log_data[2].valid := 1, [673].log_data[3].valid := 1, [673].log_data[4].valid := 1, [673].log_data[5].valid := 1, [673].log_data[6].valid := 1, [673].log_data[7].valid := 1, [673].log_data[8].valid := 1, [673].log_data[9].valid := 1, [673].log_data[10].valid := 1, [673].log_data[11].valid := 1, [673].log_data[12].valid := 1, [673].log_data[13].valid := 1, [673].log_data[14].valid := 1, [673].log_data[15].valid := 1, [673].log_data[16].valid := 1, [673].log_data[17].valid := 1, [673].log_data[18].valid := 1, [673].log_data[19].valid := 1, [673].time.Year := 2023,
        [673].time.Month := 1, [673].time.Day := 12, [673].time.Minute := 29, [673].time.Second := 59, [674].log_data[0].min := 1.0, [674].log_data[0].max := 1.0, [674].log_data[0].total := 300.0, [674].log_data[0].time := 300.0, [674].log_data[0].minminute := 30, [674].log_data[0].maxminute := 30, [674].log_data[0].valid := 1, [674].log_data[1].valid := 1, [674].log_data[2].valid := 1, [674].log_data[3].valid := 1, [674].log_data[4].valid := 1, [674].log_data[5].valid := 1, [674].log_data[6].valid := 1, [674].log_data[7].valid := 1, [674].log_data[8].valid := 1, [674].log_data[9].valid := 1, [674].log_data[10].valid := 1, [674].log_data[11].valid := 1, [674].log_data[12].valid := 1, [674].log_data[13].valid := 1, [674].log_data[14].valid := 1, [674].log_data[15].valid := 1, [674].log_data[16].valid := 1, [674].log_data[17].valid := 1, [674].log_data[18].valid := 1, [674].log_data[19].valid := 1, [674].time.Year := 2023, [674].time.Month := 1, [674].time.Day := 12, [674].time.Minute := 34, [674].time.Second := 59, [675].log_data[0].min := 1.0, [675].log_data[0].max := 1.0, [675].log_data[0].total := 300.0, [675].log_data[0].time := 300.0, [675].log_data[0].minminute := 35, [675].log_data[0].maxminute := 35, [675].log_data[0].valid := 1, [675].log_data[1].valid := 1, [675].log_data[2].valid := 1, [675].log_data[3].valid := 1, [675].log_data[4].valid := 1, [675].log_data[5].valid := 1, [675].log_data[6].valid := 1, [675].log_data[7].valid := 1, [675].log_data[8].valid := 1, [675].log_data[9].valid := 1, [675].log_data[10].valid := 1, [675].log_data[11].valid := 1, [675].log_data[12].valid := 1, [675].log_data[13].valid := 1, [675].log_data[14].valid := 1, [675].log_data[15].valid := 1, [675].log_data[16].valid := 1, [675].log_data[17].valid := 1, [675].log_data[18].valid := 1,
        [675].log_data[19].valid := 1, [675].time.Year := 2023, [675].time.Month := 1, [675].time.Day := 12, [675].time.Minute := 39, [675].time.Second := 59, [676].log_data[0].min := 1.0, [676].log_data[0].max := 1.0, [676].log_data[0].total := 300.0, [676].log_data[0].time := 300.0, [676].log_data[0].minminute := 40, [676].log_data[0].maxminute := 40, [676].log_data[0].valid := 1, [676].log_data[1].valid := 1, [676].log_data[2].valid := 1, [676].log_data[3].valid := 1, [676].log_data[4].valid := 1, [676].log_data[5].valid := 1, [676].log_data[6].valid := 1, [676].log_data[7].valid := 1, [676].log_data[8].valid := 1, [676].log_data[9].valid := 1, [676].log_data[10].valid := 1, [676].log_data[11].valid := 1, [676].log_data[12].valid := 1, [676].log_data[13].valid := 1, [676].log_data[14].valid := 1, [676].log_data[15].valid := 1, [676].log_data[16].valid := 1, [676].log_data[17].valid := 1, [676].log_data[18].valid := 1, [676].log_data[19].valid := 1, [676].time.Year := 2023, [676].time.Month := 1, [676].time.Day := 12, [676].time.Minute := 44, [676].time.Second := 59, [677].log_data[0].min := 1.0, [677].log_data[0].max := 1.0, [677].log_data[0].total := 300.0, [677].log_data[0].time := 300.0, [677].log_data[0].minminute := 45, [677].log_data[0].maxminute := 45, [677].log_data[0].valid := 1, [677].log_data[1].valid := 1, [677].log_data[2].valid := 1, [677].log_data[3].valid := 1, [677].log_data[4].valid := 1, [677].log_data[5].valid := 1, [677].log_data[6].valid := 1, [677].log_data[7].valid := 1, [677].log_data[8].valid := 1, [677].log_data[9].valid := 1, [677].log_data[10].valid := 1, [677].log_data[11].valid := 1, [677].log_data[12].valid := 1, [677].log_data[13].valid := 1, [677].log_data[14].valid := 1, [677].log_data[15].valid := 1, [677].log_data[16].valid := 1,
